  MoveL (T13838) to (110.9, 104.08, 17.5) mm, rotated rx 180 ry 0 rz -180 deg; joints [2.977, 71.493, -37.876, 5.367, -33.733, -4.467]
  MoveL (T13839) to (110.9, 104.08, 15.5) mm, rotated rx 180 ry 0 rz -180 deg; joints [2.977, 71.493, -37.876, 5.367, -33.733, -4.467]
  Set speed (40.0 mm/s)
  Call Extruder 2.0
  MoveL (T13840) to (110.9, 104.08, 15.5) mm, rotated rx 180 ry 0 rz -180 deg; joints [1.43, 67.002, -29.425, 2.343, -37.6, -1.857]
  Set speed (26.9 mm/s)
  MoveL (T13841) to (110.9, 104.08, 15.5) mm, rotated rx 180 ry 0 rz -180 deg; joints [1.43, 67.002, -29.425, 2.343, -37.6, -1.857]
  Call Extruder 0.01643
  MoveL (T13842) to (111.26, 104.43, 15.5) mm, rotated rx 180 ry 0 rz -180 deg; joints [1.43, 67.002, -29.425, 2.343, -37.6, -1.857]
  Call Extruder 0.0201
  MoveL (T13843) to (111.26, 105.05, 15.5) mm, rotated rx 180 ry 0 rz -180 deg; joints [1.431, 66.869, -29.176, 2.34, -37.717, -1.851]
  Call Extruder 0.01643
  MoveL (T13844) to (110.9, 104.69, 15.5) mm, rotated rx 180 ry 0 rz -180 deg; joints [1.431, 66.869, -29.176, 2.34, -37.717, -1.851]
  Set speed (45.0 mm/s)
  Call Extruder -1.6
  MoveL (T13845) to (110.9, 104.69, 15.5) mm, rotated rx 180 ry 0 rz -180 deg; joints [1.431, 66.869, -29.176, 2.34, -37.717, -1.851]
  Set speed (120.0 mm/s)
  MoveL (T13846) to (110.9, 104.69, 15.5) mm, rotated rx 180 ry 0 rz -180 deg; joints [3.031, 71.501, -37.892, 5.464, -33.73, -4.548]
  Call Extruder -0.17945
  MoveL (T13847) to (111.26, 105.05, 15.5) mm, rotated rx 180 ry 0 rz -180 deg; joints [3.031, 71.501, -37.892, 5.464, -33.73, -4.548]
  Call Extruder -0.20055
  MoveL (T13848) to (111.26, 104.49, 15.5) mm, rotated rx 180 ry 0 rz -180 deg; joints [3.031, 71.501, -37.892, 5.464, -33.73, -4.548]
  Set speed (45.0 mm/s)
  Call Extruder -0.02
  MoveL (T13849) to (111.26, 104.49, 15.5) mm, rotated rx 180 ry 0 rz -180 deg; joints [3.084, 71.51, -37.908, 5.56, -33.726, -4.629]
  Set speed (150.0 mm/s)
  MoveL (T13850) to (111.26, 104.49, 17.5) mm, rotated rx 180 ry 0 rz -180 deg; joints [3.084, 71.51, -37.908, 5.56, -33.726, -4.629]
  MoveL (T13851) to (117.12, 105.75, 17.5) mm, rotated rx 180 ry 0 rz -180 deg; joints [1.432, 66.737, -28.928, 2.336, -37.833, -1.845]
  MoveL (T13852) to (117.12, 105.75, 15.5) mm, rotated rx 180 ry 0 rz -180 deg; joints [1.432, 66.737, -28.928, 2.336, -37.833, -1.845]
  Set speed (40.0 mm/s)
  Call Extruder 2.0
  MoveL (T13853) to (117.12, 105.75, 15.5) mm, rotated rx 180 ry 0 rz -180 deg; joints [1.434, 66.606, -28.681, 2.332, -37.949, -1.839]
  Set speed (26.9 mm/s)
  MoveL (T13854) to (117.12, 105.75, 15.5) mm, rotated rx 180 ry 0 rz -180 deg; joints [1.434, 66.606, -28.681, 2.332, -37.949, -1.839]
  Call Extruder 0.01433
  MoveL (T13855) to (117.59, 105.75, 15.5) mm, rotated rx 180 ry 0 rz -180 deg; joints [1.434, 66.606, -28.681, 2.332, -37.949, -1.839]
  Call Extruder 0.05792
  MoveL (T13856) to (117.59, 103.84, 15.5) mm, rotated rx 180 ry 0 rz -180 deg; joints [1.434, 66.606, -28.681, 2.332, -37.949, -1.839]
  Call Extruder 0.00216
  MoveL (T13857) to (117.66, 103.84, 15.5) mm, rotated rx 180 ry 0 rz -180 deg; joints [1.434, 66.606, -28.681, 2.332, -37.949, -1.839]
  Call Extruder 0.10261
  MoveL (T13858) to (120.04, 106.23, 15.5) mm, rotated rx 180 ry 0 rz -180 deg; joints [3.137, 71.518, -37.924, 5.657, -33.723, -4.71]
  Call Extruder 0.0339
  MoveL (T13859) to (121.16, 106.23, 15.5) mm, rotated rx 180 ry 0 rz -180 deg; joints [3.137, 71.518, -37.924, 5.657, -33.723, -4.71]
  Call Extruder 0.07254
  MoveL (T13860) to (121.16, 103.84, 15.5) mm, rotated rx 180 ry 0 rz -180 deg; joints [3.137, 71.518, -37.924, 5.657, -33.723, -4.71]
  Call Extruder 0.7458
  MoveL (T13861) to (103.84, 121.16, 15.5) mm, rotated rx 180 ry 0 rz -180 deg; joints [3.19, 71.527, -37.941, 5.753, -33.72, -4.79]
  Call Extruder 0.10645
  MoveL (T13862) to (103.84, 117.66, 15.5) mm, rotated rx 180 ry 0 rz -180 deg; joints [3.19, 71.527, -37.941, 5.753, -33.72, -4.79]
  Call Extruder 0.15054
  MoveL (T13863) to (107.34, 121.16, 15.5) mm, rotated rx 180 ry 0 rz -180 deg; joints [3.19, 71.527, -37.941, 5.753, -33.72, -4.79]
  Call Extruder 0.03385
  MoveL (T13864) to (108.45, 121.16, 15.5) mm, rotated rx 180 ry 0 rz -180 deg; joints [1.435, 66.475, -28.435, 2.328, -38.064, -1.833]
  Call Extruder 0.45878
  MoveL (T13865) to (119.1, 110.51, 15.5) mm, rotated rx 180 ry 0 rz -180 deg; joints [1.435, 66.475, -28.435, 2.328, -38.064, -1.833]
  Call Extruder 0.00222
  MoveL (T13866) to (119.1, 110.43, 15.5) mm, rotated rx 180 ry 0 rz -180 deg; joints [1.435, 66.475, -28.435, 2.328, -38.064, -1.833]
  Call Extruder 0.00558
  MoveL (T13867) to (119.23, 110.3, 15.5) mm, rotated rx 180 ry 0 rz -180 deg; joints [1.436, 66.41, -28.312, 2.326, -38.121, -1.83]
  Call Extruder 0.00874
  MoveL (T13868) to (119.23, 110.02, 15.5) mm, rotated rx 180 ry 0 rz -180 deg; joints [1.436, 66.41, -28.312, 2.326, -38.121, -1.83]
  Call Extruder 0.18404
  MoveL (T13869) to (114.96, 105.75, 15.5) mm, rotated rx 180 ry 0 rz -180 deg; joints [1.436, 66.41, -28.312, 2.326, -38.121, -1.83]
  Call Extruder 0.00938
  MoveL (T13870) to (114.65, 105.75, 15.5) mm, rotated rx 180 ry 0 rz -180 deg; joints [1.436, 66.41, -28.312, 2.326, -38.121, -1.83]
  Call Extruder 0.46548
  MoveL (T13871) to (103.84, 116.55, 15.5) mm, rotated rx 180 ry 0 rz -180 deg; joints [1.436, 66.41, -28.312, 2.326, -38.121, -1.83]
  Call Extruder 0.10645
  MoveL (T13872) to (103.84, 113.06, 15.5) mm, rotated rx 180 ry 0 rz -180 deg; joints [1.463, 66.412, -28.315, 2.371, -38.12, -1.866]
  Call Extruder 0.34896
  MoveL (T13873) to (111.94, 121.16, 15.5) mm, rotated rx 180 ry 0 rz -180 deg; joints [3.218, 71.452, -37.799, 5.794, -33.788, -4.82]
  Call Extruder 0.03385
  MoveL (T13874) to (113.06, 121.16, 15.5) mm, rotated rx 180 ry 0 rz -180 deg; joints [3.221, 71.293, -37.5, 5.778, -33.928, -4.799]
  Call Extruder 0.26585
  MoveL (T13875) to (119.23, 114.98, 15.5) mm, rotated rx 180 ry 0 rz -180 deg; joints [1.518, 66.415, -28.322, 2.46, -38.119, -1.936]
  Call Extruder 0.01108
  MoveL (T13876) to (119.23, 114.62, 15.5) mm, rotated rx 180 ry 0 rz -180 deg; joints [1.518, 66.415, -28.322, 2.46, -38.119, -1.936]
  Call Extruder 0.38238
  MoveL (T13877) to (110.35, 105.75, 15.5) mm, rotated rx 180 ry 0 rz -180 deg; joints [1.518, 66.415, -28.322, 2.46, -38.119, -1.936]
  Call Extruder 0.00938
  MoveL (T13878) to (110.04, 105.75, 15.5) mm, rotated rx 180 ry 0 rz -180 deg; joints [1.573, 66.419, -28.328, 2.55, -38.118, -2.006]
  Call Extruder 0.26706
  MoveL (T13879) to (103.84, 111.94, 15.5) mm, rotated rx 180 ry 0 rz -180 deg; joints [3.224, 71.135, -37.203, 5.763, -34.067, -4.779]
  Call Extruder 0.07441
  MoveL (T13880) to (103.84, 109.5, 15.5) mm, rotated rx 180 ry 0 rz -180 deg; joints [3.224, 71.135, -37.203, 5.763, -34.067, -4.779]
  Set speed (45.0 mm/s)
  Call Extruder -1.6
  MoveL (T13881) to (103.84, 109.5, 15.5) mm, rotated rx 180 ry 0 rz -180 deg; joints [3.227, 70.978, -36.908, 5.748, -34.205, -4.758]
  Set speed (120.0 mm/s)
  MoveL (T13882) to (103.84, 109.5, 15.5) mm, rotated rx 180 ry 0 rz -180 deg; joints [3.227, 70.978, -36.908, 5.748, -34.205, -4.758]
  Call Extruder -0.38
  MoveL (T13883) to (103.84, 110.57, 15.5) mm, rotated rx 180 ry 0 rz -180 deg; joints [1.629, 66.423, -28.335, 2.639, -38.117, -2.077]
  Set speed (45.0 mm/s)
  Call Extruder -0.02
  MoveL (T13884) to (103.84, 110.57, 15.5) mm, rotated rx 180 ry 0 rz -180 deg; joints [1.629, 66.423, -28.335, 2.639, -38.117, -2.077]
  Set speed (150.0 mm/s)
  MoveL (T13885) to (103.84, 110.57, 17.5) mm, rotated rx 180 ry 0 rz -180 deg; joints [1.684, 66.426, -28.342, 2.728, -38.116, -2.147]
  MoveL (T13886) to (119.1, 110.71, 17.5) mm, rotated rx 180 ry 0 rz -180 deg; joints [1.684, 66.426, -28.342, 2.728, -38.116, -2.147]
  MoveL (T13887) to (119.1, 110.71, 15.5) mm, rotated rx 180 ry 0 rz -180 deg; joints [1.684, 66.426, -28.342, 2.728, -38.116, -2.147]
  Set speed (40.0 mm/s)
  Call Extruder 2.0
  MoveL (T13888) to (119.1, 110.71, 15.5) mm, rotated rx 180 ry 0 rz -180 deg; joints [3.23, 70.823, -36.615, 5.733, -34.342, -4.738]
  Set speed (26.9 mm/s)
  MoveL (T13889) to (119.1, 110.71, 15.5) mm, rotated rx 180 ry 0 rz -180 deg; joints [3.233, 70.668, -36.324, 5.718, -34.477, -4.719]
  Call Extruder 0.00658
  MoveL (T13890) to (119.1, 110.93, 15.5) mm, rotated rx 180 ry 0 rz -180 deg; joints [3.233, 70.668, -36.324, 5.718, -34.477, -4.719]
  Call Extruder 0.01378
  MoveL (T13891) to (119.42, 111.25, 15.5) mm, rotated rx 180 ry 0 rz -180 deg; joints [3.233, 70.668, -36.324, 5.718, -34.477, -4.719]
  Call Extruder 0.03162
  MoveL (T13892) to (120.46, 111.25, 15.5) mm, rotated rx 180 ry 0 rz -180 deg; joints [1.739, 66.43, -28.35, 2.818, -38.114, -2.217]
  Call Extruder 0.03012
  MoveL (T13893) to (121.16, 111.94, 15.5) mm, rotated rx 180 ry 0 rz -180 deg; joints [1.739, 66.43, -28.35, 2.818, -38.114, -2.217]
  Call Extruder 0.02649
  MoveL (T13894) to (121.16, 112.81, 15.5) mm, rotated rx 180 ry 0 rz -180 deg; joints [1.739, 66.43, -28.35, 2.818, -38.114, -2.217]
  Call Extruder 0.04792
  MoveL (T13895) to (119.58, 112.81, 15.5) mm, rotated rx 180 ry 0 rz -180 deg; joints [1.794, 66.434, -28.357, 2.907, -38.113, -2.288]
  Set speed (150.0 mm/s)
  MoveL (T13896) to (120.91, 113.57, 15.5) mm, rotated rx 180 ry 0 rz -180 deg; joints [1.794, 66.434, -28.357, 2.907, -38.113, -2.288]
  Set speed (26.9 mm/s)
  MoveL (T13897) to (120.91, 113.57, 15.5) mm, rotated rx 180 ry 0 rz -180 deg; joints [3.236, 70.515, -36.035, 5.704, -34.612, -4.699]
  Call Extruder 0.01626
  MoveL (T13898) to (120.56, 113.22, 15.5) mm, rotated rx 180 ry 0 rz -180 deg; joints [3.236, 70.515, -36.035, 5.704, -34.612, -4.699]
  Call Extruder 0.02045
  MoveL (T13899) to (119.94, 113.22, 15.5) mm, rotated rx 180 ry 0 rz -180 deg; joints [3.236, 70.515, -36.035, 5.704, -34.612, -4.699]
  Call Extruder 0.01626
  MoveL (T13900) to (120.29, 113.57, 15.5) mm, rotated rx 180 ry 0 rz -180 deg; joints [3.239, 70.362, -35.748, 5.69, -34.746, -4.68]
  Set speed (45.0 mm/s)
  Call Extruder -1.6
  MoveL (T13901) to (120.29, 113.57, 15.5) mm, rotated rx 180 ry 0 rz -180 deg; joints [3.239, 70.362, -35.748, 5.69, -34.746, -4.68]
  Set speed (120.0 mm/s)
  MoveL (T13902) to (120.29, 113.57, 15.5) mm, rotated rx 180 ry 0 rz -180 deg; joints [3.239, 70.362, -35.748, 5.69, -34.746, -4.68]
  Call Extruder -0.17616
  MoveL (T13903) to (119.94, 113.22, 15.5) mm, rotated rx 180 ry 0 rz -180 deg; joints [1.849, 66.438, -28.365, 2.996, -38.111, -2.358]
  Call Extruder -0.20384
  MoveL (T13904) to (120.51, 113.22, 15.5) mm, rotated rx 180 ry 0 rz -180 deg; joints [1.849, 66.438, -28.365, 2.996, -38.111, -2.358]
  Set speed (45.0 mm/s)
  Call Extruder -0.02
  MoveL (T13905) to (120.51, 113.22, 15.5) mm, rotated rx 180 ry 0 rz -180 deg; joints [1.904, 66.443, -28.373, 3.086, -38.11, -2.429]
  Set speed (150.0 mm/s)
  MoveL (T13906) to (120.51, 113.22, 17.5) mm, rotated rx 180 ry 0 rz -180 deg; joints [1.904, 66.443, -28.373, 3.086, -38.11, -2.429]
  MoveL (T13907) to (121.02, 111.02, 17.5) mm, rotated rx 180 ry 0 rz -180 deg; joints [3.242, 70.211, -35.463, 5.676, -34.88, -4.661]
  MoveL (T13908) to (121.02, 111.02, 15.5) mm, rotated rx 180 ry 0 rz -180 deg; joints [3.242, 70.211, -35.463, 5.676, -34.88, -4.661]
  Set speed (40.0 mm/s)
  Call Extruder 2.0
  MoveL (T13909) to (121.02, 111.02, 15.5) mm, rotated rx 180 ry 0 rz -180 deg; joints [3.245, 70.06, -35.18, 5.663, -35.012, -4.643]
  Set speed (26.9 mm/s)
  MoveL (T13910) to (121.02, 111.02, 15.5) mm, rotated rx 180 ry 0 rz -180 deg; joints [3.245, 70.06, -35.18, 5.663, -35.012, -4.643]
  Call Extruder 0.01707
  MoveL (T13911) to (120.64, 110.65, 15.5) mm, rotated rx 180 ry 0 rz -180 deg; joints [1.959, 66.447, -28.381, 3.175, -38.108, -2.499]
  Call Extruder 0.01989
  MoveL (T13912) to (120.03, 110.65, 15.5) mm, rotated rx 180 ry 0 rz -180 deg; joints [1.959, 66.447, -28.381, 3.175, -38.108, -2.499]
  Call Extruder 0.00867
  MoveL (T13913) to (120.22, 110.84, 15.5) mm, rotated rx 180 ry 0 rz -180 deg; joints [2.014, 66.451, -28.39, 3.264, -38.107, -2.57]
  Call Extruder 0.01989
  MoveL (T13914) to (119.61, 110.84, 15.5) mm, rotated rx 180 ry 0 rz -180 deg; joints [2.014, 66.451, -28.39, 3.264, -38.107, -2.57]
  Call Extruder 0.01299
  MoveL (T13915) to (119.32, 110.56, 15.5) mm, rotated rx 180 ry 0 rz -180 deg; joints [2.014, 66.451, -28.39, 3.264, -38.107, -2.57]
  Set speed (45.0 mm/s)
  Call Extruder -1.6
  MoveL (T13916) to (119.32, 110.56, 15.5) mm, rotated rx 180 ry 0 rz -180 deg; joints [3.248, 69.911, -34.899, 5.649, -35.143, -4.625]
  Set speed (120.0 mm/s)
  MoveL (T13917) to (119.32, 110.56, 15.5) mm, rotated rx 180 ry 0 rz -180 deg; joints [3.248, 69.911, -34.899, 5.649, -35.143, -4.625]
  Call Extruder -0.14256
  MoveL (T13918) to (119.61, 110.84, 15.5) mm, rotated rx 180 ry 0 rz -180 deg; joints [3.252, 69.762, -34.619, 5.637, -35.274, -4.607]
  Call Extruder -0.21839
  MoveL (T13919) to (120.22, 110.84, 15.5) mm, rotated rx 180 ry 0 rz -180 deg; joints [2.069, 66.456, -28.398, 3.354, -38.105, -2.64]
  Call Extruder -0.01905
  MoveL (T13920) to (120.18, 110.8, 15.5) mm, rotated rx 180 ry 0 rz -180 deg; joints [2.069, 66.456, -28.398, 3.354, -38.105, -2.64]
  Set speed (45.0 mm/s)
  Call Extruder -0.02
  MoveL (T13921) to (120.18, 110.8, 15.5) mm, rotated rx 180 ry 0 rz -180 deg; joints [2.069, 66.456, -28.398, 3.354, -38.105, -2.64]
  Set speed (150.0 mm/s)
  MoveL (T13922) to (120.18, 110.8, 17.5) mm, rotated rx 180 ry 0 rz -180 deg; joints [2.124, 66.461, -28.407, 3.443, -38.104, -2.711]
  MoveL (T13923) to (104.34, 103.54, 17.5) mm, rotated rx 180 ry 0 rz -180 deg; joints [2.124, 66.461, -28.407, 3.443, -38.104, -2.711]
  MoveL (T13924) to (104.34, 103.54, 15.7) mm, rotated rx 180 ry 0 rz -180 deg; joints [2.124, 66.461, -28.407, 3.443, -38.104, -2.711]
  Set speed (40.0 mm/s)
  Call Extruder 2.0
  MoveL (T13925) to (104.34, 103.54, 15.7) mm, rotated rx 180 ry 0 rz -180 deg; joints [3.255, 69.615, -34.341, 5.624, -35.404, -4.589]
  Set speed (26.8 mm/s)
  MoveL (T13926) to (104.34, 103.54, 15.7) mm, rotated rx 180 ry 0 rz -180 deg; joints [3.258, 69.468, -34.065, 5.611, -35.533, -4.571]
  Call Extruder 0.07908
  MoveL (T13927) to (106.94, 103.54, 15.7) mm, rotated rx 180 ry 0 rz -180 deg; joints [3.258, 69.468, -34.065, 5.611, -35.533, -4.571]
  Call Extruder 0.05792
  MoveL (T13928) to (106.93, 105.44, 15.7) mm, rotated rx 180 ry 0 rz -180 deg; joints [2.179, 66.466, -28.417, 3.533, -38.102, -2.781]
  Call Extruder 0.11363
  MoveL (T13929) to (110.66, 105.44, 15.7) mm, rotated rx 180 ry 0 rz -180 deg; joints [2.179, 66.466, -28.417, 3.533, -38.102, -2.781]
  Call Extruder 0.05792
  MoveL (T13930) to (110.67, 103.54, 15.7) mm, rotated rx 180 ry 0 rz -180 deg; joints [2.234, 66.471, -28.426, 3.622, -38.1, -2.852]
  Call Extruder 0.09209
  MoveL (T13931) to (113.69, 103.54, 15.7) mm, rotated rx 180 ry 0 rz -180 deg; joints [2.234, 66.471, -28.426, 3.622, -38.1, -2.852]
  Call Extruder 0.05792
  MoveL (T13932) to (113.69, 105.44, 15.7) mm, rotated rx 180 ry 0 rz -180 deg; joints [3.261, 69.322, -33.791, 5.599, -35.661, -4.554]
  Call Extruder 0.11347
  MoveL (T13933) to (117.41, 105.44, 15.7) mm, rotated rx 180 ry 0 rz -180 deg; joints [3.261, 69.322, -33.791, 5.599, -35.661, -4.554]
  Call Extruder 0.05792
  MoveL (T13934) to (117.41, 103.54, 15.7) mm, rotated rx 180 ry 0 rz -180 deg; joints [3.261, 69.322, -33.791, 5.599, -35.661, -4.554]
  Call Extruder 0.12333
  MoveL (T13935) to (121.46, 103.54, 15.7) mm, rotated rx 180 ry 0 rz -180 deg; joints [3.264, 69.177, -33.518, 5.587, -35.789, -4.537]
  Call Extruder 0.08749
  MoveL (T13936) to (121.46, 106.41, 15.7) mm, rotated rx 180 ry 0 rz -180 deg; joints [3.264, 69.177, -33.518, 5.587, -35.789, -4.537]
  Call Extruder 0.05864
  MoveL (T13937) to (119.54, 106.41, 15.7) mm, rotated rx 180 ry 0 rz -180 deg; joints [2.289, 66.476, -28.436, 3.712, -38.099, -2.922]
  Call Extruder 0.11623
  MoveL (T13938) to (119.53, 110.23, 15.7) mm, rotated rx 180 ry 0 rz -180 deg; joints [2.289, 66.476, -28.436, 3.712, -38.099, -2.922]
  Call Extruder 0.05869
  MoveL (T13939) to (121.46, 110.23, 15.7) mm, rotated rx 180 ry 0 rz -180 deg; joints [2.344, 66.481, -28.446, 3.801, -38.097, -2.993]
  Call Extruder 0.10898
  MoveL (T13940) to (121.46, 113.8, 15.7) mm, rotated rx 180 ry 0 rz -180 deg; joints [3.267, 69.033, -33.247, 5.575, -35.915, -4.52]
  Call Extruder 0.05874
  MoveL (T13941) to (119.53, 113.8, 15.7) mm, rotated rx 180 ry 0 rz -180 deg; joints [3.267, 69.033, -33.247, 5.575, -35.915, -4.52]
  Call Extruder 0.11558
  MoveL (T13942) to (119.53, 117.59, 15.7) mm, rotated rx 180 ry 0 rz -180 deg; joints [3.27, 68.89, -32.977, 5.563, -36.041, -4.503]
  Call Extruder 0.05879
  MoveL (T13943) to (121.46, 117.6, 15.7) mm, rotated rx 180 ry 0 rz -180 deg; joints [3.27, 68.89, -32.977, 5.563, -36.041, -4.503]
  Call Extruder 0.11768
  MoveL (T13944) to (121.46, 121.46, 15.7) mm, rotated rx 180 ry 0 rz -180 deg; joints [3.27, 68.89, -32.977, 5.563, -36.041, -4.503]
  Call Extruder 0.54596
  MoveL (T13945) to (103.54, 121.46, 15.7) mm, rotated rx 180 ry 0 rz -180 deg; joints [2.399, 66.487, -28.456, 3.89, -38.095, -3.064]
  Call Extruder 0.54596
  MoveL (T13946) to (103.54, 103.54, 15.7) mm, rotated rx 180 ry 0 rz -180 deg; joints [2.399, 66.487, -28.456, 3.89, -38.095, -3.064]
  Call Extruder 0.02254
  MoveL (T13947) to (104.28, 103.54, 15.7) mm, rotated rx 180 ry 0 rz -180 deg; joints [2.454, 66.492, -28.466, 3.98, -38.093, -3.134]
  Set speed (150.0 mm/s)
  MoveL (T13948) to (103.53, 103.13, 15.7) mm, rotated rx 180 ry 0 rz -180 deg; joints [2.454, 66.492, -28.466, 3.98, -38.093, -3.134]
  Set speed (26.8 mm/s)
  MoveL (T13949) to (103.53, 103.13, 15.7) mm, rotated rx 180 ry 0 rz -180 deg; joints [2.454, 66.492, -28.466, 3.98, -38.093, -3.134]
  Call Extruder 0.11607
  MoveL (T13950) to (107.34, 103.13, 15.7) mm, rotated rx 180 ry 0 rz -180 deg; joints [3.273, 68.747, -32.709, 5.552, -36.166, -4.487]
  Call Extruder 0.05792
  MoveL (T13951) to (107.34, 105.03, 15.7) mm, rotated rx 180 ry 0 rz -180 deg; joints [3.273, 68.747, -32.709, 5.552, -36.166, -4.487]
  Call Extruder 0.08883
  MoveL (T13952) to (110.26, 105.03, 15.7) mm, rotated rx 180 ry 0 rz -180 deg; joints [3.273, 68.747, -32.709, 5.552, -36.166, -4.487]
  Call Extruder 0.05792
  MoveL (T13953) to (110.26, 103.13, 15.7) mm, rotated rx 180 ry 0 rz -180 deg; joints [3.276, 68.606, -32.443, 5.541, -36.291, -4.471]
  Call Extruder 0.11688
  MoveL (T13954) to (114.09, 103.13, 15.7) mm, rotated rx 180 ry 0 rz -180 deg; joints [3.276, 68.606, -32.443, 5.541, -36.291, -4.471]
  Call Extruder 0.05792
  MoveL (T13955) to (114.1, 105.03, 15.7) mm, rotated rx 180 ry 0 rz -180 deg; joints [3.276, 68.606, -32.443, 5.541, -36.291, -4.471]
  Call Extruder 0.08867
  MoveL (T13956) to (117.01, 105.03, 15.7) mm, rotated rx 180 ry 0 rz -180 deg; joints [2.509, 66.498, -28.477, 4.069, -38.091, -3.205]
  Call Extruder 0.05792
  MoveL (T13957) to (117, 103.13, 15.7) mm, rotated rx 180 ry 0 rz -180 deg; joints [2.509, 66.498, -28.477, 4.069, -38.091, -3.205]
  Call Extruder 0.14814
  MoveL (T13958) to (121.87, 103.13, 15.7) mm, rotated rx 180 ry 0 rz -180 deg; joints [2.509, 66.498, -28.477, 4.069, -38.091, -3.205]
  Call Extruder 0.11229
  MoveL (T13959) to (121.87, 106.82, 15.7) mm, rotated rx 180 ry 0 rz -180 deg; joints [2.564, 66.504, -28.488, 4.159, -38.089, -3.275]
  Call Extruder 0.05865
  MoveL (T13960) to (119.94, 106.82, 15.7) mm, rotated rx 180 ry 0 rz -180 deg; joints [2.564, 66.504, -28.488, 4.159, -38.089, -3.275]
  Call Extruder 0.09143
  MoveL (T13961) to (119.94, 109.82, 15.7) mm, rotated rx 180 ry 0 rz -180 deg; joints [3.279, 68.465, -32.178, 5.53, -36.415, -4.455]
  Call Extruder 0.05869
  MoveL (T13962) to (121.87, 109.82, 15.7) mm, rotated rx 180 ry 0 rz -180 deg; joints [3.279, 68.465, -32.178, 5.53, -36.415, -4.455]
  Call Extruder 0.13381
  MoveL (T13963) to (121.87, 114.21, 15.7) mm, rotated rx 180 ry 0 rz -180 deg; joints [3.279, 68.465, -32.178, 5.53, -36.415, -4.455]
  Call Extruder 0.05875
  MoveL (T13964) to (119.94, 114.21, 15.7) mm, rotated rx 180 ry 0 rz -180 deg; joints [3.282, 68.325, -31.914, 5.519, -36.538, -4.439]
  Call Extruder 0.09077
  MoveL (T13965) to (119.94, 117.19, 15.7) mm, rotated rx 180 ry 0 rz -180 deg; joints [3.282, 68.325, -31.914, 5.519, -36.538, -4.439]
  Call Extruder 0.05879
  MoveL (T13966) to (121.87, 117.19, 15.7) mm, rotated rx 180 ry 0 rz -180 deg; joints [3.282, 68.325, -31.914, 5.519, -36.538, -4.439]
  Call Extruder 0.14247
  MoveL (T13967) to (121.87, 121.87, 15.7) mm, rotated rx 180 ry 0 rz -180 deg; joints [2.619, 66.509, -28.499, 4.248, -38.087, -3.346]
  Call Extruder 0.57077
  MoveL (T13968) to (103.13, 121.87, 15.7) mm, rotated rx 180 ry 0 rz -180 deg; joints [2.619, 66.509, -28.499, 4.248, -38.087, -3.346]
  Call Extruder 0.57077
  MoveL (T13969) to (103.13, 103.13, 15.7) mm, rotated rx 180 ry 0 rz -180 deg; joints [2.674, 66.516, -28.51, 4.338, -38.085, -3.417]
  Call Extruder 0.01036
  MoveL (T13970) to (103.47, 103.13, 15.7) mm, rotated rx 180 ry 0 rz -180 deg; joints [2.674, 66.516, -28.51, 4.338, -38.085, -3.417]
  Set speed (150.0 mm/s)
  MoveL (T13971) to (102.72, 102.81, 15.7) mm, rotated rx 180 ry 0 rz -180 deg; joints [3.285, 68.186, -31.652, 5.508, -36.66, -4.423]
  Set speed (25.0 mm/s)
  MoveL (T13972) to (102.72, 102.81, 15.7) mm, rotated rx 180 ry 0 rz -180 deg; joints [3.285, 68.186, -31.652, 5.508, -36.66, -4.423]
  Call Extruder 0.00259
  MoveL (T13973) to (102.72, 102.72, 15.7) mm, rotated rx 180 ry 0 rz -180 deg; joints [3.289, 68.047, -31.392, 5.498, -36.782, -4.408]
  Call Extruder 0.15306
  MoveL (T13974) to (107.75, 102.72, 15.7) mm, rotated rx 180 ry 0 rz -180 deg; joints [3.289, 68.047, -31.392, 5.498, -36.782, -4.408]
  Call Extruder 0.05792
  MoveL (T13975) to (107.75, 104.63, 15.7) mm, rotated rx 180 ry 0 rz -180 deg; joints [2.729, 66.522, -28.522, 4.427, -38.083, -3.488]
  Call Extruder 0.06403
  MoveL (T13976) to (109.85, 104.63, 15.7) mm, rotated rx 180 ry 0 rz -180 deg; joints [2.784, 66.528, -28.534, 4.517, -38.081, -3.558]
  Call Extruder 0.05792
  MoveL (T13977) to (109.85, 102.72, 15.7) mm, rotated rx 180 ry 0 rz -180 deg; joints [2.784, 66.528, -28.534, 4.517, -38.081, -3.558]
  Call Extruder 0.14167
  MoveL (T13978) to (114.5, 102.72, 15.7) mm, rotated rx 180 ry 0 rz -180 deg; joints [2.784, 66.528, -28.534, 4.517, -38.081, -3.558]
  Call Extruder 0.05792
  MoveL (T13979) to (114.5, 104.63, 15.7) mm, rotated rx 180 ry 0 rz -180 deg; joints [3.292, 67.909, -31.132, 5.487, -36.903, -4.393]
  Call Extruder 0.06386
  MoveL (T13980) to (116.6, 104.63, 15.7) mm, rotated rx 180 ry 0 rz -180 deg; joints [3.292, 67.909, -31.132, 5.487, -36.903, -4.393]
  Call Extruder 0.05792
  MoveL (T13981) to (116.6, 102.72, 15.7) mm, rotated rx 180 ry 0 rz -180 deg; joints [3.295, 67.772, -30.875, 5.477, -37.024, -4.378]
  Call Extruder 0.17294
  MoveL (T13982) to (122.28, 102.72, 15.7) mm, rotated rx 180 ry 0 rz -180 deg; joints [3.295, 67.772, -30.875, 5.477, -37.024, -4.378]
  Call Extruder 0.13709
  MoveL (T13983) to (122.28, 107.22, 15.7) mm, rotated rx 180 ry 0 rz -180 deg; joints [3.295, 67.772, -30.875, 5.477, -37.024, -4.378]
  Call Extruder 0.05865
  MoveL (T13984) to (120.35, 107.23, 15.7) mm, rotated rx 180 ry 0 rz -180 deg; joints [2.839, 66.534, -28.546, 4.606, -38.079, -3.629]
  Call Extruder 0.06663
  MoveL (T13985) to (120.35, 109.41, 15.7) mm, rotated rx 180 ry 0 rz -180 deg; joints [2.839, 66.534, -28.546, 4.606, -38.079, -3.629]
  Call Extruder 0.05868
  MoveL (T13986) to (122.28, 109.41, 15.7) mm, rotated rx 180 ry 0 rz -180 deg; joints [2.894, 66.541, -28.558, 4.696, -38.076, -3.7]
  Call Extruder 0.15863
  MoveL (T13987) to (122.28, 114.62, 15.7) mm, rotated rx 180 ry 0 rz -180 deg; joints [2.894, 66.541, -28.558, 4.696, -38.076, -3.7]
  Call Extruder 0.05875
  MoveL (T13988) to (120.35, 114.62, 15.7) mm, rotated rx 180 ry 0 rz -180 deg; joints [3.298, 67.636, -30.618, 5.467, -37.144, -4.363]
  Call Extruder 0.06597
  MoveL (T13989) to (120.34, 116.78, 15.7) mm, rotated rx 180 ry 0 rz -180 deg; joints [3.298, 67.636, -30.618, 5.467, -37.144, -4.363]
  Call Extruder 0.05878
  MoveL (T13990) to (122.28, 116.78, 15.7) mm, rotated rx 180 ry 0 rz -180 deg; joints [3.301, 67.5, -30.363, 5.457, -37.263, -4.348]
  Call Extruder 0.16725
  MoveL (T13991) to (122.28, 122.28, 15.7) mm, rotated rx 180 ry 0 rz -180 deg; joints [3.301, 67.5, -30.363, 5.457, -37.263, -4.348]
  Call Extruder 0.59557
  MoveL (T13992) to (102.72, 122.28, 15.7) mm, rotated rx 180 ry 0 rz -180 deg; joints [3.301, 67.5, -30.363, 5.457, -37.263, -4.348]
  Call Extruder 0.59115
  MoveL (T13993) to (102.72, 102.87, 15.7) mm, rotated rx 180 ry 0 rz -180 deg; joints [2.949, 66.548, -28.57, 4.786, -38.074, -3.771]
  Set speed (150.0 mm/s)
  MoveL (T13994) to (102.78, 102.75, 15.7) mm, rotated rx 180 ry 0 rz -180 deg; joints [2.949, 66.548, -28.57, 4.786, -38.074, -3.771]
  Set speed (45.0 mm/s)
  Call Extruder -1.6
  MoveL (T13995) to (102.78, 102.75, 15.7) mm, rotated rx 180 ry 0 rz -180 deg; joints [2.949, 66.548, -28.57, 4.786, -38.074, -3.771]
  Set speed (120.0 mm/s)
  MoveL (T13996) to (102.78, 102.75, 15.7) mm, rotated rx 180 ry 0 rz -180 deg; joints [3.004, 66.554, -28.583, 4.875, -38.072, -3.841]
  Call Extruder -0.05166
  MoveL (T13997) to (102.72, 102.72, 15.7) mm, rotated rx 180 ry 0 rz -180 deg; joints [3.004, 66.554, -28.583, 4.875, -38.072, -3.841]
  Call Extruder -0.32834
  MoveL (T13998) to (103.65, 102.72, 15.7) mm, rotated rx 180 ry 0 rz -180 deg; joints [3.004, 66.554, -28.583, 4.875, -38.072, -3.841]
  Set speed (45.0 mm/s)
  Call Extruder -0.02
  MoveL (T13999) to (103.65, 102.72, 15.7) mm, rotated rx 180 ry 0 rz -180 deg; joints [3.304, 67.365, -30.109, 5.448, -37.381, -4.334]
  Set speed (150.0 mm/s)
  MoveL (T14000) to (103.65, 102.72, 17.7) mm, rotated rx 180 ry 0 rz -180 deg; joints [3.307, 67.231, -29.857, 5.438, -37.499, -4.319]
  MoveL (T14001) to (106.29, 103.84, 17.7) mm, rotated rx 180 ry 0 rz -180 deg; joints [3.307, 67.231, -29.857, 5.438, -37.499, -4.319]
  MoveL (T14002) to (106.29, 103.84, 15.7) mm, rotated rx 180 ry 0 rz -180 deg; joints [3.059, 66.561, -28.596, 4.965, -38.07, -3.912]
  Set speed (40.0 mm/s)
  Call Extruder 2.0
  MoveL (T14003) to (106.29, 103.84, 15.7) mm, rotated rx 180 ry 0 rz -180 deg; joints [3.059, 66.561, -28.596, 4.965, -38.07, -3.912]
  Set speed (26.8 mm/s)
  MoveL (T14004) to (106.29, 103.84, 15.7) mm, rotated rx 180 ry 0 rz -180 deg; joints [3.059, 66.561, -28.596, 4.965, -38.07, -3.912]
  Call Extruder 0.07441
  MoveL (T14005) to (103.84, 103.84, 15.7) mm, rotated rx 180 ry 0 rz -180 deg; joints [3.114, 66.568, -28.61, 5.054, -38.067, -3.983]
  Call Extruder 0.7458
  MoveL (T14006) to (121.16, 121.16, 15.7) mm, rotated rx 180 ry 0 rz -180 deg; joints [3.114, 66.568, -28.61, 5.054, -38.067, -3.983]
  Call Extruder 0.09909
  MoveL (T14007) to (121.16, 117.9, 15.7) mm, rotated rx 180 ry 0 rz -180 deg; joints [3.311, 67.098, -29.605, 5.429, -37.617, -4.305]
  Call Extruder 0.00735
  MoveL (T14008) to (120.91, 117.9, 15.7) mm, rotated rx 180 ry 0 rz -180 deg; joints [3.311, 67.098, -29.605, 5.429, -37.617, -4.305]
  Call Extruder 0.14015
  MoveL (T14009) to (117.66, 121.16, 15.7) mm, rotated rx 180 ry 0 rz -180 deg; joints [3.311, 67.098, -29.605, 5.429, -37.617, -4.305]
  Call Extruder 0.03385
  MoveL (T14010) to (116.55, 121.16, 15.7) mm, rotated rx 180 ry 0 rz -180 deg; joints [3.314, 66.965, -29.355, 5.42, -37.734, -4.291]
  Call Extruder 0.54738
  MoveL (T14011) to (103.84, 108.45, 15.7) mm, rotated rx 180 ry 0 rz -180 deg; joints [3.314, 66.965, -29.355, 5.42, -37.734, -4.291]
  Call Extruder 0.03385
  MoveL (T14012) to (103.84, 107.34, 15.7) mm, rotated rx 180 ry 0 rz -180 deg; joints [3.314, 66.965, -29.355, 5.42, -37.734, -4.291]
  Call Extruder 0.11997
  MoveL (T14013) to (106.63, 104.55, 15.7) mm, rotated rx 180 ry 0 rz -180 deg; joints [3.169, 66.576, -28.623, 5.144, -38.065, -4.054]
  Call Extruder 0.0363
  MoveL (T14014) to (106.63, 105.75, 15.7) mm, rotated rx 180 ry 0 rz -180 deg; joints [3.169, 66.576, -28.623, 5.144, -38.065, -4.054]
  Call Extruder 0.03811
  MoveL (T14015) to (107.88, 105.75, 15.7) mm, rotated rx 180 ry 0 rz -180 deg; joints [3.169, 66.576, -28.623, 5.144, -38.065, -4.054]
  Set speed (45.0 mm/s)
  Call Extruder -1.6
  MoveL (T14016) to (107.88, 105.75, 15.7) mm, rotated rx 180 ry 0 rz -180 deg; joints [3.224, 66.583, -28.637, 5.234, -38.062, -4.125]
  Set speed (120.0 mm/s)
  MoveL (T14017) to (107.88, 105.75, 15.7) mm, rotated rx 180 ry 0 rz -180 deg; joints [3.224, 66.583, -28.637, 5.234, -38.062, -4.125]
  Call Extruder -0.38
  MoveL (T14018) to (106.81, 105.75, 15.7) mm, rotated rx 180 ry 0 rz -180 deg; joints [3.224, 66.583, -28.637, 5.234, -38.062, -4.125]
  Set speed (45.0 mm/s)
  Call Extruder -0.02
  MoveL (T14019) to (106.81, 105.75, 15.7) mm, rotated rx 180 ry 0 rz -180 deg; joints [3.317, 66.833, -29.107, 5.411, -37.85, -4.277]
  Set speed (150.0 mm/s)
  MoveL (T14020) to (106.81, 105.75, 17.7) mm, rotated rx 180 ry 0 rz -180 deg; joints [3.317, 66.833, -29.107, 5.411, -37.85, -4.277]
  MoveL (T14021) to (110.61, 105.75, 17.7) mm, rotated rx 180 ry 0 rz -180 deg; joints [3.317, 66.833, -29.107, 5.411, -37.85, -4.277]
  MoveL (T14022) to (110.61, 105.75, 15.7) mm, rotated rx 180 ry 0 rz -180 deg; joints [3.317, 66.833, -29.107, 5.411, -37.85, -4.277]
  Set speed (40.0 mm/s)
  Call Extruder 2.0
  MoveL (T14023) to (110.61, 105.75, 15.7) mm, rotated rx 180 ry 0 rz -180 deg; joints [3.32, 66.701, -28.859, 5.402, -37.966, -4.264]
  Set speed (26.8 mm/s)
  MoveL (T14024) to (110.61, 105.75, 15.7) mm, rotated rx 180 ry 0 rz -180 deg; joints [3.32, 66.701, -28.859, 5.402, -37.966, -4.264]
  Call Extruder 0.00593
  MoveL (T14025) to (110.75, 105.87, 15.7) mm, rotated rx 180 ry 0 rz -180 deg; joints [3.262, 66.547, -28.569, 5.292, -38.097, -4.169]
  Call Extruder 0.01451
  MoveL (T14026) to (111.23, 105.87, 15.7) mm, rotated rx 180 ry 0 rz -180 deg; joints [3.262, 66.547, -28.569, 5.292, -38.097, -4.169]
  Call Extruder 0.01375
  MoveL (T14027) to (111.55, 105.55, 15.7) mm, rotated rx 180 ry 0 rz -180 deg; joints [3.262, 66.547, -28.569, 5.292, -38.097, -4.169]
  Call Extruder 0.04007
  MoveL (T14028) to (111.55, 104.24, 15.7) mm, rotated rx 180 ry 0 rz -180 deg; joints [3.262, 66.547, -28.569, 5.292, -38.097, -4.169]
  Call Extruder 0.01698
  MoveL (T14029) to (111.94, 103.84, 15.7) mm, rotated rx 180 ry 0 rz -180 deg; joints [3.262, 66.547, -28.569, 5.292, -38.097, -4.169]
  Call Extruder 0.02453
  MoveL (T14030) to (112.75, 103.84, 15.7) mm, rotated rx 180 ry 0 rz -180 deg; joints [3.262, 66.547, -28.569, 5.292, -38.097, -4.169]
  Call Extruder 0.04988
  MoveL (T14031) to (112.75, 105.48, 15.7) mm, rotated rx 180 ry 0 rz -180 deg; joints [3.262, 66.547, -28.569, 5.292, -38.097, -4.169]
  Set speed (150.0 mm/s)
  MoveL (T14032) to (113.57, 104.67, 15.7) mm, rotated rx 180 ry 0 rz -180 deg; joints [3.262, 66.547, -28.569, 5.292, -38.097, -4.169]
  Set speed (26.8 mm/s)
  MoveL (T14033) to (113.57, 104.67, 15.7) mm, rotated rx 180 ry 0 rz -180 deg; joints [3.262, 66.547, -28.569, 5.292, -38.097, -4.169]
  Call Extruder 0.01928
  MoveL (T14034) to (113.16, 105.08, 15.7) mm, rotated rx 180 ry 0 rz -180 deg; joints [3.32, 66.701, -28.859, 5.402, -37.966, -4.264]
  Call Extruder 0.02098
  MoveL (T14035) to (113.16, 104.45, 15.7) mm, rotated rx 180 ry 0 rz -180 deg; joints [3.32, 66.701, -28.859, 5.402, -37.966, -4.264]
  Call Extruder 0.01928
  MoveL (T14036) to (113.57, 104.05, 15.7) mm, rotated rx 180 ry 0 rz -180 deg; joints [3.318, 66.77, -28.989, 5.407, -37.905, -4.271]
  Set speed (45.0 mm/s)
  Call Extruder -1.6
  MoveL (T14037) to (113.57, 104.05, 15.7) mm, rotated rx 180 ry 0 rz -180 deg; joints [3.318, 66.77, -28.989, 5.407, -37.905, -4.271]
  Set speed (120.0 mm/s)
  MoveL (T14038) to (113.57, 104.05, 15.7) mm, rotated rx 180 ry 0 rz -180 deg; joints [3.318, 66.77, -28.989, 5.407, -37.905, -4.271]
  Call Extruder -0.20613
  MoveL (T14039) to (113.16, 104.45, 15.7) mm, rotated rx 180 ry 0 rz -180 deg; joints [3.318, 66.77, -28.989, 5.407, -37.905, -4.271]
  Call Extruder -0.17387
  MoveL (T14040) to (113.16, 104.94, 15.7) mm, rotated rx 180 ry 0 rz -180 deg; joints [3.318, 66.77, -28.989, 5.407, -37.905, -4.271]
  Set speed (45.0 mm/s)
  Call Extruder -0.02
  MoveL (T14041) to (113.16, 104.94, 15.7) mm, rotated rx 180 ry 0 rz -180 deg; joints [3.318, 66.77, -28.989, 5.407, -37.905, -4.271]
  Set speed (150.0 mm/s)
  MoveL (T14042) to (113.16, 104.94, 17.7) mm, rotated rx 180 ry 0 rz -180 deg; joints [3.318, 66.77, -28.989, 5.407, -37.905, -4.271]
  MoveL (T14043) to (110.86, 105.65, 17.7) mm, rotated rx 180 ry 0 rz -180 deg; joints [3.318, 66.532, -28.948, 5.431, -37.709, -4.301]
  MoveL (T14044) to (110.86, 105.65, 15.7) mm, rotated rx 180 ry 0 rz -180 deg; joints [3.318, 66.532, -28.948, 5.431, -37.709, -4.301]
  Set speed (40.0 mm/s)
  Call Extruder 2.0
  MoveL (T14045) to (110.86, 105.65, 15.7) mm, rotated rx 180 ry 0 rz -180 deg; joints [3.318, 66.532, -28.948, 5.431, -37.709, -4.301]
  Set speed (26.8 mm/s)
  MoveL (T14046) to (110.86, 105.65, 15.7) mm, rotated rx 180 ry 0 rz -180 deg; joints [3.318, 66.532, -28.948, 5.431, -37.709, -4.301]
  Call Extruder 0.01251
  MoveL (T14047) to (111.14, 105.37, 15.7) mm, rotated rx 180 ry 0 rz -180 deg; joints [3.318, 66.532, -28.948, 5.431, -37.709, -4.301]
  Call Extruder 0.01919
  MoveL (T14048) to (111.14, 104.77, 15.7) mm, rotated rx 180 ry 0 rz -180 deg; joints [3.318, 66.532, -28.948, 5.431, -37.709, -4.301]
  Call Extruder 0.00781
  MoveL (T14049) to (110.97, 104.94, 15.7) mm, rotated rx 180 ry 0 rz -180 deg; joints [3.82, 66.607, -29.089, 6.256, -37.683, -4.959]
  Call Extruder 0.01919
  MoveL (T14050) to (110.97, 104.34, 15.7) mm, rotated rx 180 ry 0 rz -180 deg; joints [3.82, 66.821, -29.126, 6.231, -37.86, -4.927]
  Call Extruder 0.01606
  MoveL (T14051) to (111.33, 103.98, 15.7) mm, rotated rx 180 ry 0 rz -180 deg; joints [3.82, 66.821, -29.126, 6.231, -37.86, -4.927]
  Set speed (45.0 mm/s)
  Call Extruder -1.6
  MoveL (T14052) to (111.33, 103.98, 15.7) mm, rotated rx 180 ry 0 rz -180 deg; joints [3.82, 66.821, -29.126, 6.231, -37.86, -4.927]
  Set speed (120.0 mm/s)
  MoveL (T14053) to (111.33, 103.98, 15.7) mm, rotated rx 180 ry 0 rz -180 deg; joints [3.82, 66.821, -29.126, 6.231, -37.86, -4.927]
  Call Extruder -0.17962
  MoveL (T14054) to (110.97, 104.34, 15.7) mm, rotated rx 180 ry 0 rz -180 deg; joints [3.82, 66.821, -29.126, 6.231, -37.86, -4.927]
  Call Extruder -0.20038
  MoveL (T14055) to (110.97, 104.9, 15.7) mm, rotated rx 180 ry 0 rz -180 deg; joints [3.82, 66.821, -29.126, 6.231, -37.86, -4.927]
  Set speed (45.0 mm/s)
  Call Extruder -0.02
  MoveL (T14056) to (110.97, 104.9, 15.7) mm, rotated rx 180 ry 0 rz -180 deg; joints [3.82, 66.821, -29.126, 6.231, -37.86, -4.927]
  Set speed (150.0 mm/s)
  MoveL (T14057) to (110.97, 104.9, 17.7) mm, rotated rx 180 ry 0 rz -180 deg; joints [3.82, 66.821, -29.126, 6.231, -37.86, -4.927]
  MoveL (T14058) to (117.12, 105.75, 17.7) mm, rotated rx 180 ry 0 rz -180 deg; joints [3.82, 66.821, -29.126, 6.231, -37.86, -4.927]
  MoveL (T14059) to (117.12, 105.75, 15.7) mm, rotated rx 180 ry 0 rz -180 deg; joints [3.82, 66.821, -29.126, 6.231, -37.86, -4.927]
  Set speed (40.0 mm/s)
  Call Extruder 2.0
  MoveL (T14060) to (117.12, 105.75, 15.7) mm, rotated rx 180 ry 0 rz -180 deg; joints [3.834, 66.317, -28.177, 6.193, -38.303, -4.867]
  Set speed (26.8 mm/s)
  MoveL (T14061) to (117.12, 105.75, 15.7) mm, rotated rx 180 ry 0 rz -180 deg; joints [3.834, 66.317, -28.177, 6.193, -38.303, -4.867]
  Call Extruder 0.01822
  MoveL (T14062) to (117.72, 105.75, 15.7) mm, rotated rx 180 ry 0 rz -180 deg; joints [3.803, 65.911, -27.413, 6.095, -38.656, -4.766]
  Call Extruder 0.05619
  MoveL (T14063) to (117.72, 103.9, 15.7) mm, rotated rx 180 ry 0 rz -180 deg; joints [3.803, 65.911, -27.413, 6.095, -38.656, -4.766]
  Call Extruder 0.09501
  MoveL (T14064) to (119.92, 106.11, 15.7) mm, rotated rx 180 ry 0 rz -180 deg; joints [3.803, 65.911, -27.413, 6.095, -38.656, -4.766]
  Call Extruder 0.03754
  MoveL (T14065) to (121.16, 106.11, 15.7) mm, rotated rx 180 ry 0 rz -180 deg; joints [3.693, 65.591, -26.813, 5.883, -38.926, -4.583]
  Call Extruder 0.0689
  MoveL (T14066) to (121.16, 103.84, 15.7) mm, rotated rx 180 ry 0 rz -180 deg; joints [3.693, 65.591, -26.813, 5.883, -38.926, -4.583]
  Call Extruder 0.7458
  MoveL (T14067) to (103.84, 121.16, 15.7) mm, rotated rx 180 ry 0 rz -180 deg; joints [3.693, 65.591, -26.813, 5.883, -38.926, -4.583]
  Call Extruder 0.10645
  MoveL (T14068) to (103.84, 117.66, 15.7) mm, rotated rx 180 ry 0 rz -180 deg; joints [3.493, 65.421, -26.492, 5.548, -39.06, -4.313]
  Call Extruder 0.15054
  MoveL (T14069) to (107.34, 121.16, 15.7) mm, rotated rx 180 ry 0 rz -180 deg; joints [3.493, 65.421, -26.492, 5.548, -39.06, -4.313]
  Call Extruder 0.03385
  MoveL (T14070) to (108.45, 121.16, 15.7) mm, rotated rx 180 ry 0 rz -180 deg; joints [1.308, 65.214, -26.103, 2.072, -39.129, -1.608]
  Call Extruder 0.45879
  MoveL (T14071) to (119.1, 110.51, 15.7) mm, rotated rx 180 ry 0 rz -180 deg; joints [1.308, 65.214, -26.103, 2.072, -39.129, -1.608]
  Call Extruder 0.00577
  MoveL (T14072) to (119.1, 110.32, 15.7) mm, rotated rx 180 ry 0 rz -180 deg; joints [1.134, 65.303, -26.27, 1.801, -39.046, -1.399]
  Call Extruder 0.00558
  MoveL (T14073) to (119.23, 110.19, 15.7) mm, rotated rx 180 ry 0 rz -180 deg; joints [1, 65.567, -26.767, 1.596, -38.811, -1.244]
  Call Extruder 0.00516
  MoveL (T14074) to (119.23, 110.02, 15.7) mm, rotated rx 180 ry 0 rz -180 deg; joints [1, 65.567, -26.767, 1.596, -38.811, -1.244]
  Call Extruder 0.18405
  MoveL (T14075) to (114.96, 105.75, 15.7) mm, rotated rx 180 ry 0 rz -180 deg; joints [1, 65.567, -26.767, 1.596, -38.811, -1.244]
  Call Extruder 0.00939
  MoveL (T14076) to (114.65, 105.75, 15.7) mm, rotated rx 180 ry 0 rz -180 deg; joints [0.934, 66.034, -27.646, 1.505, -38.398, -1.179]
  Call Extruder 0.46547
  MoveL (T14077) to (103.84, 116.55, 15.7) mm, rotated rx 180 ry 0 rz -180 deg; joints [0.934, 66.034, -27.646, 1.505, -38.398, -1.179]
  Call Extruder 0.10645
  MoveL (T14078) to (103.84, 113.06, 15.7) mm, rotated rx 180 ry 0 rz -180 deg; joints [0.934, 66.034, -27.646, 1.505, -38.398, -1.179]
  Call Extruder 0.34896
  MoveL (T14079) to (111.94, 121.16, 15.7) mm, rotated rx 180 ry 0 rz -180 deg; joints [0.9, 71.665, -38.239, 1.634, -33.436, -1.364]
  Call Extruder 0.03385
  MoveL (T14080) to (113.06, 121.16, 15.7) mm, rotated rx 180 ry 0 rz -180 deg; joints [0.9, 71.665, -38.239, 1.634, -33.436, -1.364]
  Call Extruder 0.26587
  MoveL (T14081) to (119.23, 114.98, 15.7) mm, rotated rx 180 ry 0 rz -180 deg; joints [0.939, 72.175, -39.199, 1.725, -32.988, -1.447]
  Call Extruder 0.01106
  MoveL (T14082) to (119.23, 114.62, 15.7) mm, rotated rx 180 ry 0 rz -180 deg; joints [0.939, 72.175, -39.199, 1.725, -32.988, -1.447]
  Call Extruder 0.38238
  MoveL (T14083) to (110.35, 105.75, 15.7) mm, rotated rx 180 ry 0 rz -180 deg; joints [1.05, 72.578, -39.958, 1.948, -32.635, -1.641]
  Call Extruder 0.00939
  MoveL (T14084) to (110.04, 105.75, 15.7) mm, rotated rx 180 ry 0 rz -180 deg; joints [1.05, 72.578, -39.958, 1.948, -32.635, -1.641]
  Call Extruder 0.26705
  MoveL (T14085) to (103.84, 111.94, 15.7) mm, rotated rx 180 ry 0 rz -180 deg; joints [1.244, 72.781, -40.34, 2.318, -32.462, -1.956]
  Call Extruder 0.07441
  MoveL (T14086) to (103.84, 109.5, 15.7) mm, rotated rx 180 ry 0 rz -180 deg; joints [1.244, 72.781, -40.34, 2.318, -32.462, -1.956]
  Set speed (45.0 mm/s)
  Call Extruder -1.6
  MoveL (T14087) to (103.84, 109.5, 15.7) mm, rotated rx 180 ry 0 rz -180 deg; joints [3.323, 73.051, -40.847, 6.219, -32.356, -5.259]
  Set speed (120.0 mm/s)
  MoveL (T14088) to (103.84, 109.5, 15.7) mm, rotated rx 180 ry 0 rz -180 deg; joints [3.323, 73.051, -40.847, 6.219, -32.356, -5.259]
  Call Extruder -0.38
  MoveL (T14089) to (103.84, 110.57, 15.7) mm, rotated rx 180 ry 0 rz -180 deg; joints [3.49, 72.949, -40.656, 6.512, -32.461, -5.501]
  Set speed (45.0 mm/s)
  Call Extruder -0.02
  MoveL (T14090) to (103.84, 110.57, 15.7) mm, rotated rx 180 ry 0 rz -180 deg; joints [3.49, 72.949, -40.656, 6.512, -32.461, -5.501]
  Set speed (150.0 mm/s)
  MoveL (T14091) to (103.84, 110.57, 17.7) mm, rotated rx 180 ry 0 rz -180 deg; joints [3.622, 72.609, -40.016, 6.702, -32.771, -5.643]
  MoveL (T14092) to (119.1, 110.71, 17.7) mm, rotated rx 180 ry 0 rz -180 deg; joints [3.622, 72.609, -40.016, 6.702, -32.771, -5.643]
  MoveL (T14093) to (119.1, 110.71, 15.7) mm, rotated rx 180 ry 0 rz -180 deg; joints [3.694, 72.008, -38.886, 6.738, -33.305, -5.64]
  Set speed (40.0 mm/s)
  Call Extruder 2.0
  MoveL (T14094) to (119.1, 110.71, 15.7) mm, rotated rx 180 ry 0 rz -180 deg; joints [3.694, 72.008, -38.886, 6.738, -33.305, -5.64]
  Set speed (26.8 mm/s)
  MoveL (T14095) to (119.1, 110.71, 15.7) mm, rotated rx 180 ry 0 rz -180 deg; joints [3.819, 66.837, -29.155, 6.233, -37.846, -4.929]
  Call Extruder 0.00302
  MoveL (T14096) to (119.1, 110.81, 15.7) mm, rotated rx 180 ry 0 rz -180 deg; joints [3.819, 66.837, -29.155, 6.233, -37.846, -4.929]
  Call Extruder 0.01378
  MoveL (T14097) to (119.42, 111.13, 15.7) mm, rotated rx 180 ry 0 rz -180 deg; joints [3.819, 66.837, -29.155, 6.233, -37.846, -4.929]
  Call Extruder 0.02805
  MoveL (T14098) to (120.34, 111.13, 15.7) mm, rotated rx 180 ry 0 rz -180 deg; joints [3.819, 66.837, -29.155, 6.233, -37.846, -4.929]
  Call Extruder 0.03515
  MoveL (T14099) to (121.16, 111.94, 15.7) mm, rotated rx 180 ry 0 rz -180 deg; joints [3.819, 66.837, -29.155, 6.233, -37.846, -4.929]
  Call Extruder 0.02988
  MoveL (T14100) to (121.16, 112.92, 15.7) mm, rotated rx 180 ry 0 rz -180 deg; joints [3.819, 66.837, -29.155, 6.233, -37.846, -4.929]
  Call Extruder 0.04453
  MoveL (T14101) to (119.69, 112.92, 15.7) mm, rotated rx 180 ry 0 rz -180 deg; joints [3.819, 66.837, -29.155, 6.233, -37.846, -4.929]
  Set speed (150.0 mm/s)
  MoveL (T14102) to (121, 113.15, 15.7) mm, rotated rx 180 ry 0 rz -180 deg; joints [3.819, 66.837, -29.155, 6.233, -37.846, -4.929]
  Set speed (26.8 mm/s)
  MoveL (T14103) to (121, 113.15, 15.7) mm, rotated rx 180 ry 0 rz -180 deg; joints [3.827, 66.561, -28.636, 6.211, -38.088, -4.896]
  Call Extruder 0.01587
  MoveL (T14104) to (120.65, 113.5, 15.7) mm, rotated rx 180 ry 0 rz -180 deg; joints [3.827, 66.561, -28.636, 6.211, -38.088, -4.896]
  Call Extruder 0.01955
  MoveL (T14105) to (120.04, 113.5, 15.7) mm, rotated rx 180 ry 0 rz -180 deg; joints [3.827, 66.561, -28.636, 6.211, -38.088, -4.896]
  Call Extruder 0.00755
  MoveL (T14106) to (120.21, 113.33, 15.7) mm, rotated rx 180 ry 0 rz -180 deg; joints [3.827, 66.561, -28.636, 6.211, -38.088, -4.896]
  Call Extruder 0.01955
  MoveL (T14107) to (119.6, 113.33, 15.7) mm, rotated rx 180 ry 0 rz -180 deg; joints [3.827, 66.561, -28.636, 6.211, -38.088, -4.896]
  Call Extruder 0.01276
  MoveL (T14108) to (119.32, 113.61, 15.7) mm, rotated rx 180 ry 0 rz -180 deg; joints [1.407, 66.288, -28.531, 2.298, -37.78, -1.816]
  Set speed (45.0 mm/s)
  Call Extruder -1.6
  MoveL (T14109) to (119.32, 113.61, 15.7) mm, rotated rx 180 ry 0 rz -180 deg; joints [1.407, 66.526, -28.571, 2.287, -37.977, -1.803]
  Set speed (120.0 mm/s)
  MoveL (T14110) to (119.32, 113.61, 15.7) mm, rotated rx 180 ry 0 rz -180 deg; joints [1.407, 66.526, -28.571, 2.287, -37.977, -1.803]
  Call Extruder -0.14126
  MoveL (T14111) to (119.6, 113.33, 15.7) mm, rotated rx 180 ry 0 rz -180 deg; joints [1.407, 66.526, -28.571, 2.287, -37.977, -1.803]
  Call Extruder -0.21639
  MoveL (T14112) to (120.21, 113.33, 15.7) mm, rotated rx 180 ry 0 rz -180 deg; joints [1.407, 66.526, -28.571, 2.287, -37.977, -1.803]
  Call Extruder -0.02235
  MoveL (T14113) to (120.17, 113.38, 15.7) mm, rotated rx 180 ry 0 rz -180 deg; joints [1.407, 66.526, -28.571, 2.287, -37.977, -1.803]
  Set speed (45.0 mm/s)
  Call Extruder -0.02
  MoveL (T14114) to (120.17, 113.38, 15.7) mm, rotated rx 180 ry 0 rz -180 deg; joints [1.407, 66.526, -28.571, 2.287, -37.977, -1.803]
  Set speed (150.0 mm/s)
  MoveL (T14115) to (120.17, 113.38, 17.7) mm, rotated rx 180 ry 0 rz -180 deg; joints [1.363, 71.364, -37.673, 2.456, -33.715, -2.044]
  MoveL (T14116) to (120.92, 110.35, 17.7) mm, rotated rx 180 ry 0 rz -180 deg; joints [1.363, 71.364, -37.673, 2.456, -33.715, -2.044]
  MoveL (T14117) to (120.92, 110.35, 15.7) mm, rotated rx 180 ry 0 rz -180 deg; joints [3.241, 71.591, -38.101, 5.86, -33.629, -4.884]
  Set speed (40.0 mm/s)
  Call Extruder 2.0
  MoveL (T14118) to (120.92, 110.35, 15.7) mm, rotated rx 180 ry 0 rz -180 deg; joints [3.351, 66.512, -28.544, 5.437, -38.093, -4.284]
  Set speed (26.8 mm/s)
  MoveL (T14119) to (120.92, 110.35, 15.7) mm, rotated rx 180 ry 0 rz -180 deg; joints [3.351, 66.512, -28.544, 5.437, -38.093, -4.284]
  Call Extruder 0.01747
  MoveL (T14120) to (120.55, 110.72, 15.7) mm, rotated rx 180 ry 0 rz -180 deg; joints [1.409, 66.321, -28.185, 2.282, -38.158, -1.794]
  Call Extruder 0.0208
  MoveL (T14121) to (119.92, 110.72, 15.7) mm, rotated rx 180 ry 0 rz -180 deg; joints [1.409, 66.321, -28.185, 2.282, -38.158, -1.794]
  Call Extruder 0.01747
  MoveL (T14122) to (120.3, 110.35, 15.7) mm, rotated rx 180 ry 0 rz -180 deg; joints [1.407, 66.511, -28.542, 2.287, -37.991, -1.803]
  Set speed (45.0 mm/s)
  Call Extruder -1.6
  MoveL (T14123) to (120.3, 110.35, 15.7) mm, rotated rx 180 ry 0 rz -180 deg; joints [1.407, 66.511, -28.542, 2.287, -37.991, -1.803]
  Set speed (120.0 mm/s)
  MoveL (T14124) to (120.3, 110.35, 15.7) mm, rotated rx 180 ry 0 rz -180 deg; joints [1.365, 66.317, -28.177, 2.21, -38.16, -1.738]
  Call Extruder -0.18758
  MoveL (T14125) to (119.92, 110.72, 15.7) mm, rotated rx 180 ry 0 rz -180 deg; joints [1.365, 66.317, -28.177, 2.21, -38.16, -1.738]
  Call Extruder -0.19242
  MoveL (T14126) to (120.46, 110.72, 15.7) mm, rotated rx 180 ry 0 rz -180 deg; joints [1.365, 66.317, -28.177, 2.21, -38.16, -1.738]
  Set speed (45.0 mm/s)
  Call Extruder -0.02
  MoveL (T14127) to (120.46, 110.72, 15.7) mm, rotated rx 180 ry 0 rz -180 deg; joints [1.365, 66.317, -28.177, 2.21, -38.16, -1.738]
  Set speed (150.0 mm/s)
  MoveL (T14128) to (120.46, 110.72, 17.7) mm, rotated rx 180 ry 0 rz -180 deg; joints [1.365, 66.317, -28.177, 2.21, -38.16, -1.738]
  MoveL (T14129) to (104.34, 103.54, 17.7) mm, rotated rx 180 ry 0 rz -180 deg; joints [1.365, 66.317, -28.177, 2.21, -38.16, -1.738]
  MoveL (T14130) to (104.34, 103.54, 15.9) mm, rotated rx 180 ry 0 rz -180 deg; joints [1.319, 71.489, -37.909, 2.385, -33.603, -1.986]
  Set speed (40.0 mm/s)
  Call Extruder 2.0
  MoveL (T14131) to (104.34, 103.54, 15.9) mm, rotated rx 180 ry 0 rz -180 deg; joints [1.319, 71.489, -37.909, 2.385, -33.603, -1.986]
  Set speed (26.8 mm/s)
  MoveL (T14132) to (104.34, 103.54, 15.9) mm, rotated rx 180 ry 0 rz -180 deg; joints [3.282, 71.728, -38.358, 5.951, -33.512, -4.967]
  Call Extruder 0.07565
  MoveL (T14133) to (106.82, 103.54, 15.9) mm, rotated rx 180 ry 0 rz -180 deg; joints [3.398, 66.414, -28.36, 5.502, -38.183, -4.33]
  Call Extruder 0.05793
  MoveL (T14134) to (106.82, 105.44, 15.9) mm, rotated rx 180 ry 0 rz -180 deg; joints [3.398, 66.414, -28.36, 5.502, -38.183, -4.33]
  Call Extruder 0.11362
  MoveL (T14135) to (110.55, 105.44, 15.9) mm, rotated rx 180 ry 0 rz -180 deg; joints [3.398, 66.414, -28.36, 5.502, -38.183, -4.33]
  Call Extruder 0.05793
  MoveL (T14136) to (110.55, 103.54, 15.9) mm, rotated rx 180 ry 0 rz -180 deg; joints [1.366, 66.215, -27.985, 2.207, -38.25, -1.734]
  Call Extruder 0.09938
  MoveL (T14137) to (113.81, 103.54, 15.9) mm, rotated rx 180 ry 0 rz -180 deg; joints [1.366, 66.215, -27.985, 2.207, -38.25, -1.734]
  Call Extruder 0.05793
  MoveL (T14138) to (113.81, 105.44, 15.9) mm, rotated rx 180 ry 0 rz -180 deg; joints [1.365, 66.301, -28.148, 2.21, -38.174, -1.737]
  Call Extruder 0.11352
  MoveL (T14139) to (117.54, 105.44, 15.9) mm, rotated rx 180 ry 0 rz -180 deg; joints [1.365, 66.301, -28.148, 2.21, -38.174, -1.737]
  Call Extruder 0.05793
  MoveL (T14140) to (117.54, 103.54, 15.9) mm, rotated rx 180 ry 0 rz -180 deg; joints [1.365, 66.301, -28.148, 2.21, -38.174, -1.737]
  Call Extruder 0.11943
  MoveL (T14141) to (121.46, 103.54, 15.9) mm, rotated rx 180 ry 0 rz -180 deg; joints [1.365, 66.301, -28.148, 2.21, -38.174, -1.737]
  Call Extruder 0.08385
  MoveL (T14142) to (121.46, 106.29, 15.9) mm, rotated rx 180 ry 0 rz -180 deg; joints [1.332, 66.109, -27.787, 2.148, -38.342, -1.685]
  Call Extruder 0.05863
  MoveL (T14143) to (119.54, 106.29, 15.9) mm, rotated rx 180 ry 0 rz -180 deg; joints [1.332, 66.109, -27.787, 2.148, -38.342, -1.685]
  Call Extruder 0.11631
  MoveL (T14144) to (119.53, 110.11, 15.9) mm, rotated rx 180 ry 0 rz -180 deg; joints [1.332, 66.109, -27.787, 2.148, -38.342, -1.685]
  Call Extruder 0.05868
  MoveL (T14145) to (121.46, 110.11, 15.9) mm, rotated rx 180 ry 0 rz -180 deg; joints [1.332, 66.109, -27.787, 2.148, -38.342, -1.685]
  Call Extruder 0.11593
  MoveL (T14146) to (121.46, 113.92, 15.9) mm, rotated rx 180 ry 0 rz -180 deg; joints [1.332, 66.109, -27.787, 2.148, -38.342, -1.685]
  Call Extruder 0.05873
  MoveL (T14147) to (119.53, 113.91, 15.9) mm, rotated rx 180 ry 0 rz -180 deg; joints [1.323, 66.109, -27.786, 2.133, -38.342, -1.673]
  Call Extruder 0.11564
  MoveL (T14148) to (119.53, 117.71, 15.9) mm, rotated rx 180 ry 0 rz -180 deg; joints [1.276, 71.615, -38.145, 2.313, -33.491, -1.929]
  Call Extruder 0.05879
  MoveL (T14149) to (121.46, 117.71, 15.9) mm, rotated rx 180 ry 0 rz -180 deg; joints [3.322, 71.865, -38.617, 6.043, -33.395, -5.051]
  Call Extruder 0.11423
  MoveL (T14150) to (121.46, 121.46, 15.9) mm, rotated rx 180 ry 0 rz -180 deg; joints [3.322, 71.865, -38.617, 6.043, -33.395, -5.051]
  Call Extruder 0.54596
  MoveL (T14151) to (103.54, 121.46, 15.9) mm, rotated rx 180 ry 0 rz -180 deg; joints [3.445, 66.316, -28.176, 5.566, -38.272, -4.375]
  Call Extruder 0.54596
  MoveL (T14152) to (103.54, 103.54, 15.9) mm, rotated rx 180 ry 0 rz -180 deg; joints [3.445, 66.316, -28.176, 5.566, -38.272, -4.375]
  Call Extruder 0.02254
  MoveL (T14153) to (104.28, 103.54, 15.9) mm, rotated rx 180 ry 0 rz -180 deg; joints [3.445, 66.316, -28.176, 5.566, -38.272, -4.375]
  Set speed (150.0 mm/s)
  MoveL (T14154) to (103.53, 103.13, 15.9) mm, rotated rx 180 ry 0 rz -180 deg; joints [1.339, 66.11, -27.788, 2.159, -38.342, -1.693]
  Set speed (26.8 mm/s)
  MoveL (T14155) to (103.53, 103.13, 15.9) mm, rotated rx 180 ry 0 rz -180 deg; joints [1.339, 66.11, -27.788, 2.159, -38.342, -1.693]
  Call Extruder 0.11264
  MoveL (T14156) to (107.23, 103.13, 15.9) mm, rotated rx 180 ry 0 rz -180 deg; joints [1.339, 66.11, -27.788, 2.159, -38.342, -1.693]
  Call Extruder 0.05793
  MoveL (T14157) to (107.23, 105.03, 15.9) mm, rotated rx 180 ry 0 rz -180 deg; joints [1.326, 66.124, -27.815, 2.138, -38.328, -1.678]
  Call Extruder 0.08882
  MoveL (T14158) to (110.14, 105.03, 15.9) mm, rotated rx 180 ry 0 rz -180 deg; joints [1.326, 66.124, -27.815, 2.138, -38.328, -1.678]
  Call Extruder 0.05793
  MoveL (T14159) to (110.14, 103.13, 15.9) mm, rotated rx 180 ry 0 rz -180 deg; joints [1.326, 66.124, -27.815, 2.138, -38.328, -1.678]
  Call Extruder 0.12417
  MoveL (T14160) to (114.22, 103.13, 15.9) mm, rotated rx 180 ry 0 rz -180 deg; joints [1.326, 66.124, -27.815, 2.138, -38.328, -1.678]
  Call Extruder 0.05793
  MoveL (T14161) to (114.22, 105.03, 15.9) mm, rotated rx 180 ry 0 rz -180 deg; joints [1.326, 66.124, -27.815, 2.138, -38.328, -1.678]
  Call Extruder 0.08871
  MoveL (T14162) to (117.13, 105.03, 15.9) mm, rotated rx 180 ry 0 rz -180 deg; joints [1.326, 66.124, -27.815, 2.138, -38.328, -1.678]
  Call Extruder 0.05793
  MoveL (T14163) to (117.13, 103.13, 15.9) mm, rotated rx 180 ry 0 rz -180 deg; joints [1.326, 66.124, -27.815, 2.138, -38.328, -1.678]
  Call Extruder 0.14424
  MoveL (T14164) to (121.87, 103.13, 15.9) mm, rotated rx 180 ry 0 rz -180 deg; joints [1.326, 66.124, -27.815, 2.138, -38.328, -1.678]
  Call Extruder 0.10865
  MoveL (T14165) to (121.87, 106.7, 15.9) mm, rotated rx 180 ry 0 rz -180 deg; joints [1.326, 66.124, -27.815, 2.138, -38.328, -1.678]
  Call Extruder 0.05864
  MoveL (T14166) to (119.94, 106.7, 15.9) mm, rotated rx 180 ry 0 rz -180 deg; joints [1.326, 66.124, -27.815, 2.138, -38.328, -1.678]
  Call Extruder 0.09151
  MoveL (T14167) to (119.94, 109.7, 15.9) mm, rotated rx 180 ry 0 rz -180 deg; joints [1.323, 66.109, -27.786, 2.133, -38.342, -1.673]
  Call Extruder 0.05868
  MoveL (T14168) to (121.87, 109.7, 15.9) mm, rotated rx 180 ry 0 rz -180 deg; joints [1.321, 66.344, -28.228, 2.139, -38.135, -1.683]
  Call Extruder 0.14076
  MoveL (T14169) to (121.87, 114.32, 15.9) mm, rotated rx 180 ry 0 rz -180 deg; joints [1.321, 66.344, -28.228, 2.139, -38.135, -1.683]
  Call Extruder 0.05874
  MoveL (T14170) to (119.94, 114.32, 15.9) mm, rotated rx 180 ry 0 rz -180 deg; joints [1.321, 66.344, -28.228, 2.139, -38.135, -1.683]
  Call Extruder 0.09084
  MoveL (T14171) to (119.94, 117.3, 15.9) mm, rotated rx 180 ry 0 rz -180 deg; joints [1.321, 66.344, -28.228, 2.139, -38.135, -1.683]
  Call Extruder 0.05878
  MoveL (T14172) to (121.87, 117.31, 15.9) mm, rotated rx 180 ry 0 rz -180 deg; joints [1.321, 66.344, -28.228, 2.139, -38.135, -1.683]
  Call Extruder 0.13901
  MoveL (T14173) to (121.87, 121.87, 15.9) mm, rotated rx 180 ry 0 rz -180 deg; joints [1.321, 66.344, -28.228, 2.139, -38.135, -1.683]
  Call Extruder 0.57077
  MoveL (T14174) to (103.13, 121.87, 15.9) mm, rotated rx 180 ry 0 rz -180 deg; joints [1.321, 66.344, -28.228, 2.139, -38.135, -1.683]
  Call Extruder 0.57077
  MoveL (T14175) to (103.13, 103.13, 15.9) mm, rotated rx 180 ry 0 rz -180 deg; joints [1.321, 66.105, -28.188, 2.149, -37.937, -1.695]
  Call Extruder 0.01036
  MoveL (T14176) to (103.47, 103.13, 15.9) mm, rotated rx 180 ry 0 rz -180 deg; joints [3.142, 71.301, -37.949, 5.702, -33.483, -4.761]
  Set speed (150.0 mm/s)
  MoveL (T14177) to (102.72, 102.81, 15.9) mm, rotated rx 180 ry 0 rz -180 deg; joints [3.142, 71.536, -37.997, 5.674, -33.669, -4.727]
  Set speed (25.0 mm/s)
  MoveL (T14178) to (102.72, 102.81, 15.9) mm, rotated rx 180 ry 0 rz -180 deg; joints [3.142, 71.536, -37.997, 5.674, -33.669, -4.727]
  Call Extruder 0.00259
  MoveL (T14179) to (102.72, 102.72, 15.9) mm, rotated rx 180 ry 0 rz -180 deg; joints [3.142, 71.536, -37.997, 5.674, -33.669, -4.727]
  Call Extruder 0.14964
  MoveL (T14180) to (107.64, 102.72, 15.9) mm, rotated rx 180 ry 0 rz -180 deg; joints [3.142, 71.536, -37.997, 5.674, -33.669, -4.727]
  Call Extruder 0.05793
  MoveL (T14181) to (107.64, 104.63, 15.9) mm, rotated rx 180 ry 0 rz -180 deg; joints [3.142, 71.536, -37.997, 5.674, -33.669, -4.727]
  Call Extruder 0.06401
  MoveL (T14182) to (109.74, 104.63, 15.9) mm, rotated rx 180 ry 0 rz -180 deg; joints [3.142, 71.536, -37.997, 5.674, -33.669, -4.727]
  Call Extruder 0.05793
  MoveL (T14183) to (109.74, 102.72, 15.9) mm, rotated rx 180 ry 0 rz -180 deg; joints [3.142, 71.536, -37.997, 5.674, -33.669, -4.727]
  Call Extruder 0.14896
  MoveL (T14184) to (114.63, 102.72, 15.9) mm, rotated rx 180 ry 0 rz -180 deg; joints [3.142, 71.536, -37.997, 5.674, -33.669, -4.727]
  Call Extruder 0.05793
  MoveL (T14185) to (114.63, 104.63, 15.9) mm, rotated rx 180 ry 0 rz -180 deg; joints [3.142, 71.536, -37.997, 5.674, -33.669, -4.727]
  Call Extruder 0.06391
  MoveL (T14186) to (116.73, 104.63, 15.9) mm, rotated rx 180 ry 0 rz -180 deg; joints [3.214, 71.343, -37.635, 5.778, -33.844, -4.804]
  Call Extruder 0.05793
  MoveL (T14187) to (116.73, 102.72, 15.9) mm, rotated rx 180 ry 0 rz -180 deg; joints [3.214, 71.343, -37.635, 5.778, -33.844, -4.804]
  Call Extruder 0.16905
  MoveL (T14188) to (122.28, 102.72, 15.9) mm, rotated rx 180 ry 0 rz -180 deg; joints [3.214, 71.343, -37.635, 5.778, -33.844, -4.804]
  Call Extruder 0.13344
  MoveL (T14189) to (122.28, 107.11, 15.9) mm, rotated rx 180 ry 0 rz -180 deg; joints [3.214, 71.343, -37.635, 5.778, -33.844, -4.804]
  Call Extruder 0.05864
  MoveL (T14190) to (120.35, 107.11, 15.9) mm, rotated rx 180 ry 0 rz -180 deg; joints [3.217, 71.162, -37.294, 5.76, -34.003, -4.78]
  Call Extruder 0.06671
  MoveL (T14191) to (120.35, 109.3, 15.9) mm, rotated rx 180 ry 0 rz -180 deg; joints [3.217, 71.162, -37.294, 5.76, -34.003, -4.78]
  Call Extruder 0.05867
  MoveL (T14192) to (122.28, 109.3, 15.9) mm, rotated rx 180 ry 0 rz -180 deg; joints [3.217, 71.162, -37.294, 5.76, -34.003, -4.78]
  Call Extruder 0.16558
  MoveL (T14193) to (122.28, 114.73, 15.9) mm, rotated rx 180 ry 0 rz -180 deg; joints [3.102, 71.471, -37.875, 5.593, -33.722, -4.657]
  Call Extruder 0.05875
  MoveL (T14194) to (120.35, 114.73, 15.9) mm, rotated rx 180 ry 0 rz -180 deg; joints [3.041, 71.461, -37.857, 5.483, -33.726, -4.564]
  Call Extruder 0.06604
  MoveL (T14195) to (120.35, 116.9, 15.9) mm, rotated rx 180 ry 0 rz -180 deg; joints [3.041, 71.461, -37.857, 5.483, -33.726, -4.564]
  Call Extruder 0.05877
  MoveL (T14196) to (122.28, 116.9, 15.9) mm, rotated rx 180 ry 0 rz -180 deg; joints [3.041, 71.461, -37.857, 5.483, -33.726, -4.564]
  Call Extruder 0.1638
  MoveL (T14197) to (122.28, 122.28, 15.9) mm, rotated rx 180 ry 0 rz -180 deg; joints [3.221, 70.983, -36.956, 5.743, -34.161, -4.757]
  Call Extruder 0.59557
  MoveL (T14198) to (102.72, 122.28, 15.9) mm, rotated rx 180 ry 0 rz -180 deg; joints [3.221, 70.983, -36.956, 5.743, -34.161, -4.757]
  Call Extruder 0.59115
  MoveL (T14199) to (102.72, 102.87, 15.9) mm, rotated rx 180 ry 0 rz -180 deg; joints [3.221, 70.983, -36.956, 5.743, -34.161, -4.757]
  Set speed (150.0 mm/s)
  MoveL (T14200) to (102.78, 102.75, 15.9) mm, rotated rx 180 ry 0 rz -180 deg; joints [3.224, 70.805, -36.621, 5.726, -34.317, -4.734]
  Set speed (45.0 mm/s)
  Call Extruder -1.6
  MoveL (T14201) to (102.78, 102.75, 15.9) mm, rotated rx 180 ry 0 rz -180 deg; joints [3.224, 70.805, -36.621, 5.726, -34.317, -4.734]
  Set speed (120.0 mm/s)
  MoveL (T14202) to (102.78, 102.75, 15.9) mm, rotated rx 180 ry 0 rz -180 deg; joints [2.98, 71.452, -37.839, 5.372, -33.73, -4.472]
  Call Extruder -0.05166
  MoveL (T14203) to (102.72, 102.72, 15.9) mm, rotated rx 180 ry 0 rz -180 deg; joints [2.98, 71.452, -37.839, 5.372, -33.73, -4.472]
  Call Extruder -0.32834
  MoveL (T14204) to (103.65, 102.72, 15.9) mm, rotated rx 180 ry 0 rz -180 deg; joints [2.919, 71.442, -37.821, 5.262, -33.733, -4.38]
  Set speed (45.0 mm/s)
  Call Extruder -0.02
  MoveL (T14205) to (103.65, 102.72, 15.9) mm, rotated rx 180 ry 0 rz -180 deg; joints [2.919, 71.442, -37.821, 5.262, -33.733, -4.38]
  Set speed (150.0 mm/s)
  MoveL (T14206) to (103.65, 102.72, 17.9) mm, rotated rx 180 ry 0 rz -180 deg; joints [2.919, 71.442, -37.821, 5.262, -33.733, -4.38]
  MoveL (T14207) to (106.29, 103.84, 17.9) mm, rotated rx 180 ry 0 rz -180 deg; joints [3.228, 70.628, -36.288, 5.709, -34.473, -4.711]
  MoveL (T14208) to (106.29, 103.84, 15.9) mm, rotated rx 180 ry 0 rz -180 deg; joints [3.228, 70.628, -36.288, 5.709, -34.473, -4.711]
  Set speed (40.0 mm/s)
  Call Extruder 2.0
  MoveL (T14209) to (106.29, 103.84, 15.9) mm, rotated rx 180 ry 0 rz -180 deg; joints [3.231, 70.453, -35.959, 5.693, -34.627, -4.689]
  Set speed (26.8 mm/s)
  MoveL (T14210) to (106.29, 103.84, 15.9) mm, rotated rx 180 ry 0 rz -180 deg; joints [3.231, 70.453, -35.959, 5.693, -34.627, -4.689]
  Call Extruder 0.07441
  MoveL (T14211) to (103.84, 103.84, 15.9) mm, rotated rx 180 ry 0 rz -180 deg; joints [2.858, 71.433, -37.804, 5.152, -33.737, -4.288]
  Call Extruder 0.7458
  MoveL (T14212) to (121.16, 121.16, 15.9) mm, rotated rx 180 ry 0 rz -180 deg; joints [2.858, 71.433, -37.804, 5.152, -33.737, -4.288]
  Call Extruder 0.09564
  MoveL (T14213) to (121.16, 118.02, 15.9) mm, rotated rx 180 ry 0 rz -180 deg; joints [2.797, 71.424, -37.787, 5.041, -33.74, -4.195]
  Call Extruder 0.0108
  MoveL (T14214) to (120.8, 118.02, 15.9) mm, rotated rx 180 ry 0 rz -180 deg; joints [2.797, 71.424, -37.787, 5.041, -33.74, -4.195]
  Call Extruder 0.13527
  MoveL (T14215) to (117.66, 121.16, 15.9) mm, rotated rx 180 ry 0 rz -180 deg; joints [3.235, 70.279, -35.631, 5.677, -34.779, -4.668]
  Call Extruder 0.03385
  MoveL (T14216) to (116.55, 121.16, 15.9) mm, rotated rx 180 ry 0 rz -180 deg; joints [3.235, 70.279, -35.631, 5.677, -34.779, -4.668]
  Call Extruder 0.54738
  MoveL (T14217) to (103.84, 108.45, 15.9) mm, rotated rx 180 ry 0 rz -180 deg; joints [3.238, 70.106, -35.306, 5.661, -34.931, -4.646]
  Call Extruder 0.03385
  MoveL (T14218) to (103.84, 107.34, 15.9) mm, rotated rx 180 ry 0 rz -180 deg; joints [3.238, 70.106, -35.306, 5.661, -34.931, -4.646]
  Call Extruder 0.11512
  MoveL (T14219) to (106.52, 104.67, 15.9) mm, rotated rx 180 ry 0 rz -180 deg; joints [3.238, 70.106, -35.306, 5.661, -34.931, -4.646]
  Call Extruder 0.03288
  MoveL (T14220) to (106.52, 105.75, 15.9) mm, rotated rx 180 ry 0 rz -180 deg; joints [2.737, 71.415, -37.77, 4.931, -33.744, -4.103]
  Call Extruder 0.04153
  MoveL (T14221) to (107.88, 105.75, 15.9) mm, rotated rx 180 ry 0 rz -180 deg; joints [2.737, 71.415, -37.77, 4.931, -33.744, -4.103]
  Set speed (45.0 mm/s)
  Call Extruder -1.6
  MoveL (T14222) to (107.88, 105.75, 15.9) mm, rotated rx 180 ry 0 rz -180 deg; joints [2.676, 71.407, -37.754, 4.82, -33.747, -4.011]
  Set speed (120.0 mm/s)
  MoveL (T14223) to (107.88, 105.75, 15.9) mm, rotated rx 180 ry 0 rz -180 deg; joints [2.676, 71.407, -37.754, 4.82, -33.747, -4.011]
  Call Extruder -0.38
  MoveL (T14224) to (106.81, 105.75, 15.9) mm, rotated rx 180 ry 0 rz -180 deg; joints [3.242, 69.935, -34.984, 5.646, -35.082, -4.625]
  Set speed (45.0 mm/s)
  Call Extruder -0.02
  MoveL (T14225) to (106.81, 105.75, 15.9) mm, rotated rx 180 ry 0 rz -180 deg; joints [3.242, 69.935, -34.984, 5.646, -35.082, -4.625]
  Set speed (150.0 mm/s)
  MoveL (T14226) to (106.81, 105.75, 17.9) mm, rotated rx 180 ry 0 rz -180 deg; joints [3.242, 69.935, -34.984, 5.646, -35.082, -4.625]
  MoveL (T14227) to (110.54, 105.78, 17.9) mm, rotated rx 180 ry 0 rz -180 deg; joints [3.245, 69.765, -34.664, 5.631, -35.232, -4.605]
  MoveL (T14228) to (110.54, 105.78, 15.9) mm, rotated rx 180 ry 0 rz -180 deg; joints [3.245, 69.765, -34.664, 5.631, -35.232, -4.605]
  Set speed (40.0 mm/s)
  Call Extruder 2.0
  MoveL (T14229) to (110.54, 105.78, 15.9) mm, rotated rx 180 ry 0 rz -180 deg; joints [2.615, 71.398, -37.738, 4.71, -33.75, -3.919]
  Set speed (26.8 mm/s)
  MoveL (T14230) to (110.54, 105.78, 15.9) mm, rotated rx 180 ry 0 rz -180 deg; joints [2.615, 71.398, -37.738, 4.71, -33.75, -3.919]
  Call Extruder 0.00424
  MoveL (T14231) to (110.64, 105.87, 15.9) mm, rotated rx 180 ry 0 rz -180 deg; joints [2.615, 71.398, -37.738, 4.71, -33.75, -3.919]
  Call Extruder 0.01452
  MoveL (T14232) to (111.12, 105.87, 15.9) mm, rotated rx 180 ry 0 rz -180 deg; joints [2.615, 71.398, -37.738, 4.71, -33.75, -3.919]
  Call Extruder 0.01375
  MoveL (T14233) to (111.44, 105.55, 15.9) mm, rotated rx 180 ry 0 rz -180 deg; joints [2.554, 71.39, -37.722, 4.6, -33.753, -3.827]
  Call Extruder 0.03663
  MoveL (T14234) to (111.44, 104.35, 15.9) mm, rotated rx 180 ry 0 rz -180 deg; joints [2.554, 71.39, -37.722, 4.6, -33.753, -3.827]
  Call Extruder 0.02185
  MoveL (T14235) to (111.94, 103.84, 15.9) mm, rotated rx 180 ry 0 rz -180 deg; joints [2.554, 71.39, -37.722, 4.6, -33.753, -3.827]
  Call Extruder 0.02837
  MoveL (T14236) to (112.88, 103.84, 15.9) mm, rotated rx 180 ry 0 rz -180 deg; joints [3.249, 69.596, -34.346, 5.617, -35.38, -4.584]
  Call Extruder 0.04603
  MoveL (T14237) to (112.88, 105.36, 15.9) mm, rotated rx 180 ry 0 rz -180 deg; joints [3.249, 69.596, -34.346, 5.617, -35.38, -4.584]
  Set speed (150.0 mm/s)
  MoveL (T14238) to (113.1, 103.95, 15.9) mm, rotated rx 180 ry 0 rz -180 deg; joints [3.249, 69.596, -34.346, 5.617, -35.38, -4.584]
  Set speed (26.8 mm/s)
  MoveL (T14239) to (113.1, 103.95, 15.9) mm, rotated rx 180 ry 0 rz -180 deg; joints [3.252, 69.428, -34.03, 5.602, -35.528, -4.564]
  Call Extruder 0.01886
  MoveL (T14240) to (113.51, 104.36, 15.9) mm, rotated rx 180 ry 0 rz -180 deg; joints [3.252, 69.428, -34.03, 5.602, -35.528, -4.564]
  Call Extruder 0.02005
  MoveL (T14241) to (113.51, 104.98, 15.9) mm, rotated rx 180 ry 0 rz -180 deg; joints [2.493, 71.382, -37.707, 4.49, -33.756, -3.735]
  Call Extruder 0.01042
  MoveL (T14242) to (113.28, 104.75, 15.9) mm, rotated rx 180 ry 0 rz -180 deg; joints [2.493, 71.382, -37.707, 4.49, -33.756, -3.735]
  Call Extruder 0.02005
  MoveL (T14243) to (113.28, 105.37, 15.9) mm, rotated rx 180 ry 0 rz -180 deg; joints [2.493, 71.382, -37.707, 4.49, -33.756, -3.735]
  Call Extruder 0.01308
  MoveL (T14244) to (113.57, 105.65, 15.9) mm, rotated rx 180 ry 0 rz -180 deg; joints [2.493, 71.382, -37.707, 4.49, -33.756, -3.735]
  Set speed (45.0 mm/s)
  Call Extruder -1.6
  MoveL (T14245) to (113.57, 105.65, 15.9) mm, rotated rx 180 ry 0 rz -180 deg; joints [2.432, 71.374, -37.693, 4.38, -33.759, -3.643]
  Set speed (120.0 mm/s)
  MoveL (T14246) to (113.57, 105.65, 15.9) mm, rotated rx 180 ry 0 rz -180 deg; joints [2.432, 71.374, -37.693, 4.38, -33.759, -3.643]
  Call Extruder -0.14307
  MoveL (T14247) to (113.28, 105.37, 15.9) mm, rotated rx 180 ry 0 rz -180 deg; joints [3.256, 69.261, -33.716, 5.588, -35.674, -4.545]
  Call Extruder -0.21934
  MoveL (T14248) to (113.28, 104.75, 15.9) mm, rotated rx 180 ry 0 rz -180 deg; joints [3.256, 69.261, -33.716, 5.588, -35.674, -4.545]
  Call Extruder -0.01759
  MoveL (T14249) to (113.32, 104.78, 15.9) mm, rotated rx 180 ry 0 rz -180 deg; joints [3.256, 69.261, -33.716, 5.588, -35.674, -4.545]
  Set speed (45.0 mm/s)
  Call Extruder -0.02
  MoveL (T14250) to (113.32, 104.78, 15.9) mm, rotated rx 180 ry 0 rz -180 deg; joints [3.259, 69.096, -33.405, 5.575, -35.82, -4.525]
  Set speed (150.0 mm/s)
  MoveL (T14251) to (113.32, 104.78, 17.9) mm, rotated rx 180 ry 0 rz -180 deg; joints [3.259, 69.096, -33.405, 5.575, -35.82, -4.525]
  MoveL (T14252) to (110.67, 104.08, 17.9) mm, rotated rx 180 ry 0 rz -180 deg; joints [2.371, 71.367, -37.678, 4.269, -33.762, -3.551]
  MoveL (T14253) to (110.67, 104.08, 15.9) mm, rotated rx 180 ry 0 rz -180 deg; joints [2.371, 71.367, -37.678, 4.269, -33.762, -3.551]
  Set speed (40.0 mm/s)
  Call Extruder 2.0
  MoveL (T14254) to (110.67, 104.08, 15.9) mm, rotated rx 180 ry 0 rz -180 deg; joints [2.371, 71.367, -37.678, 4.269, -33.762, -3.551]
  Set speed (26.8 mm/s)
  MoveL (T14255) to (110.67, 104.08, 15.9) mm, rotated rx 180 ry 0 rz -180 deg; joints [2.31, 71.359, -37.664, 4.159, -33.765, -3.46]
  Call Extruder 0.01643
  MoveL (T14256) to (111.03, 104.43, 15.9) mm, rotated rx 180 ry 0 rz -180 deg; joints [2.31, 71.359, -37.664, 4.159, -33.765, -3.46]
  Call Extruder 0.0201
  MoveL (T14257) to (111.03, 105.05, 15.9) mm, rotated rx 180 ry 0 rz -180 deg; joints [3.263, 68.932, -33.096, 5.561, -35.964, -4.506]
  Call Extruder 0.01643
  MoveL (T14258) to (110.67, 104.69, 15.9) mm, rotated rx 180 ry 0 rz -180 deg; joints [3.263, 68.932, -33.096, 5.561, -35.964, -4.506]
  Set speed (45.0 mm/s)
  Call Extruder -1.6
  MoveL (T14259) to (110.67, 104.69, 15.9) mm, rotated rx 180 ry 0 rz -180 deg; joints [3.263, 68.932, -33.096, 5.561, -35.964, -4.506]
  Set speed (120.0 mm/s)
  MoveL (T14260) to (110.67, 104.69, 15.9) mm, rotated rx 180 ry 0 rz -180 deg; joints [3.266, 68.768, -32.789, 5.548, -36.108, -4.487]
  Call Extruder -0.17945
  MoveL (T14261) to (111.03, 105.05, 15.9) mm, rotated rx 180 ry 0 rz -180 deg; joints [3.266, 68.768, -32.789, 5.548, -36.108, -4.487]
  Call Extruder -0.20055
  MoveL (T14262) to (111.03, 104.49, 15.9) mm, rotated rx 180 ry 0 rz -180 deg; joints [3.266, 68.768, -32.789, 5.548, -36.108, -4.487]
  Set speed (45.0 mm/s)
  Call Extruder -0.02
  MoveL (T14263) to (111.03, 104.49, 15.9) mm, rotated rx 180 ry 0 rz -180 deg; joints [2.249, 71.352, -37.65, 4.049, -33.768, -3.368]
  Set speed (150.0 mm/s)
  MoveL (T14264) to (111.03, 104.49, 17.9) mm, rotated rx 180 ry 0 rz -180 deg; joints [2.249, 71.352, -37.65, 4.049, -33.768, -3.368]
  MoveL (T14265) to (117.12, 105.75, 17.9) mm, rotated rx 180 ry 0 rz -180 deg; joints [2.249, 71.352, -37.65, 4.049, -33.768, -3.368]
  MoveL (T14266) to (117.12, 105.75, 15.9) mm, rotated rx 180 ry 0 rz -180 deg; joints [2.188, 71.345, -37.637, 3.939, -33.77, -3.276]
  Set speed (40.0 mm/s)
  Call Extruder 2.0
  MoveL (T14267) to (117.12, 105.75, 15.9) mm, rotated rx 180 ry 0 rz -180 deg; joints [2.188, 71.345, -37.637, 3.939, -33.77, -3.276]
  Set speed (26.8 mm/s)
  MoveL (T14268) to (117.12, 105.75, 15.9) mm, rotated rx 180 ry 0 rz -180 deg; joints [3.27, 68.606, -32.484, 5.535, -36.25, -4.469]
  Call Extruder 0.02211
  MoveL (T14269) to (117.85, 105.75, 15.9) mm, rotated rx 180 ry 0 rz -180 deg; joints [3.27, 68.606, -32.484, 5.535, -36.25, -4.469]
  Call Extruder 0.0523
  MoveL (T14270) to (117.85, 104.03, 15.9) mm, rotated rx 180 ry 0 rz -180 deg; joints [3.273, 68.445, -32.18, 5.522, -36.392, -4.45]
  Call Extruder 0.08435
  MoveL (T14271) to (119.8, 105.99, 15.9) mm, rotated rx 180 ry 0 rz -180 deg; joints [3.273, 68.445, -32.18, 5.522, -36.392, -4.45]
  Call Extruder 0.04118
  MoveL (T14272) to (121.16, 105.99, 15.9) mm, rotated rx 180 ry 0 rz -180 deg; joints [2.127, 71.338, -37.624, 3.829, -33.773, -3.184]
  Call Extruder 0.06525
  MoveL (T14273) to (121.16, 103.84, 15.9) mm, rotated rx 180 ry 0 rz -180 deg; joints [2.127, 71.338, -37.624, 3.829, -33.773, -3.184]
  Call Extruder 0.7458
  MoveL (T14274) to (103.84, 121.16, 15.9) mm, rotated rx 180 ry 0 rz -180 deg; joints [2.127, 71.338, -37.624, 3.829, -33.773, -3.184]
  Call Extruder 0.10645
  MoveL (T14275) to (103.84, 117.66, 15.9) mm, rotated rx 180 ry 0 rz -180 deg; joints [2.067, 71.331, -37.612, 3.719, -33.775, -3.093]
  Call Extruder 0.15054
  MoveL (T14276) to (107.34, 121.16, 15.9) mm, rotated rx 180 ry 0 rz -180 deg; joints [2.067, 71.331, -37.612, 3.719, -33.775, -3.093]
  Call Extruder 0.03385
  MoveL (T14277) to (108.45, 121.16, 15.9) mm, rotated rx 180 ry 0 rz -180 deg; joints [3.277, 68.285, -31.88, 5.51, -36.532, -4.432]
  Call Extruder 0.45881
  MoveL (T14278) to (119.1, 110.51, 15.9) mm, rotated rx 180 ry 0 rz -180 deg; joints [3.277, 68.285, -31.88, 5.51, -36.532, -4.432]
  Call Extruder 0.00933
  MoveL (T14279) to (119.1, 110.2, 15.9) mm, rotated rx 180 ry 0 rz -180 deg; joints [3.277, 68.285, -31.88, 5.51, -36.532, -4.432]
  Call Extruder 0.00558
  MoveL (T14280) to (119.23, 110.07, 15.9) mm, rotated rx 180 ry 0 rz -180 deg; joints [3.28, 68.126, -31.58, 5.498, -36.672, -4.414]
  Call Extruder 0.00159
  MoveL (T14281) to (119.23, 110.02, 15.9) mm, rotated rx 180 ry 0 rz -180 deg; joints [3.28, 68.126, -31.58, 5.498, -36.672, -4.414]
  Call Extruder 0.18406
  MoveL (T14282) to (114.96, 105.75, 15.9) mm, rotated rx 180 ry 0 rz -180 deg; joints [2.006, 71.325, -37.6, 3.609, -33.778, -3.001]
  Call Extruder 0.0094
  MoveL (T14283) to (114.65, 105.75, 15.9) mm, rotated rx 180 ry 0 rz -180 deg; joints [2.006, 71.325, -37.6, 3.609, -33.778, -3.001]
  Call Extruder 0.46547
  MoveL (T14284) to (103.84, 116.55, 15.9) mm, rotated rx 180 ry 0 rz -180 deg; joints [1.945, 71.319, -37.588, 3.499, -33.78, -2.91]
  Call Extruder 0.10645
  MoveL (T14285) to (103.84, 113.06, 15.9) mm, rotated rx 180 ry 0 rz -180 deg; joints [1.945, 71.319, -37.588, 3.499, -33.78, -2.91]
  Call Extruder 0.34896
  MoveL (T14286) to (111.94, 121.16, 15.9) mm, rotated rx 180 ry 0 rz -180 deg; joints [1.945, 71.319, -37.588, 3.499, -33.78, -2.91]
  Call Extruder 0.03385
  MoveL (T14287) to (113.06, 121.16, 15.9) mm, rotated rx 180 ry 0 rz -180 deg; joints [3.284, 67.968, -31.283, 5.486, -36.811, -4.397]
  Call Extruder 0.26588
  MoveL (T14288) to (119.23, 114.98, 15.9) mm, rotated rx 180 ry 0 rz -180 deg; joints [3.284, 67.968, -31.283, 5.486, -36.811, -4.397]
  Call Extruder 0.01104
  MoveL (T14289) to (119.23, 114.62, 15.9) mm, rotated rx 180 ry 0 rz -180 deg; joints [3.284, 67.968, -31.283, 5.486, -36.811, -4.397]
  Call Extruder 0.38239
  MoveL (T14290) to (110.35, 105.75, 15.9) mm, rotated rx 180 ry 0 rz -180 deg; joints [3.287, 67.811, -30.987, 5.474, -36.949, -4.38]
  Call Extruder 0.0094
  MoveL (T14291) to (110.04, 105.75, 15.9) mm, rotated rx 180 ry 0 rz -180 deg; joints [3.287, 67.811, -30.987, 5.474, -36.949, -4.38]
  Call Extruder 0.26705
  MoveL (T14292) to (103.84, 111.94, 15.9) mm, rotated rx 180 ry 0 rz -180 deg; joints [3.287, 67.811, -30.987, 5.474, -36.949, -4.38]
  Call Extruder 0.07441
  MoveL (T14293) to (103.84, 109.5, 15.9) mm, rotated rx 180 ry 0 rz -180 deg; joints [1.884, 71.313, -37.576, 3.389, -33.783, -2.818]
  Set speed (45.0 mm/s)
  Call Extruder -1.6
  MoveL (T14294) to (103.84, 109.5, 15.9) mm, rotated rx 180 ry 0 rz -180 deg; joints [1.884, 71.313, -37.576, 3.389, -33.783, -2.818]
  Set speed (120.0 mm/s)
  MoveL (T14295) to (103.84, 109.5, 15.9) mm, rotated rx 180 ry 0 rz -180 deg; joints [1.884, 71.313, -37.576, 3.389, -33.783, -2.818]
  Call Extruder -0.38
  MoveL (T14296) to (103.84, 110.57, 15.9) mm, rotated rx 180 ry 0 rz -180 deg; joints [1.823, 71.307, -37.565, 3.279, -33.785, -2.726]
  Set speed (45.0 mm/s)
  Call Extruder -0.02
  MoveL (T14297) to (103.84, 110.57, 15.9) mm, rotated rx 180 ry 0 rz -180 deg; joints [1.823, 71.307, -37.565, 3.279, -33.785, -2.726]
  Set speed (150.0 mm/s)
  MoveL (T14298) to (103.84, 110.57, 17.9) mm, rotated rx 180 ry 0 rz -180 deg; joints [3.291, 67.654, -30.693, 5.463, -37.087, -4.363]
  MoveL (T14299) to (119.81, 113.03, 17.9) mm, rotated rx 180 ry 0 rz -180 deg; joints [3.291, 67.654, -30.693, 5.463, -37.087, -4.363]
  MoveL (T14300) to (119.81, 113.03, 15.9) mm, rotated rx 180 ry 0 rz -180 deg; joints [3.291, 67.654, -30.693, 5.463, -37.087, -4.363]
  Set speed (40.0 mm/s)
  Call Extruder 2.0
  MoveL (T14301) to (119.81, 113.03, 15.9) mm, rotated rx 180 ry 0 rz -180 deg; joints [3.291, 67.654, -30.693, 5.463, -37.087, -4.363]
  Set speed (26.8 mm/s)
  MoveL (T14302) to (119.81, 113.03, 15.9) mm, rotated rx 180 ry 0 rz -180 deg; joints [3.295, 67.499, -30.401, 5.452, -37.223, -4.346]
  Call Extruder 0.04114
  MoveL (T14303) to (121.16, 113.04, 15.9) mm, rotated rx 180 ry 0 rz -180 deg; joints [3.295, 67.499, -30.401, 5.452, -37.223, -4.346]
  Call Extruder 0.03327
  MoveL (T14304) to (121.16, 111.94, 15.9) mm, rotated rx 180 ry 0 rz -180 deg; joints [3.295, 67.499, -30.401, 5.452, -37.223, -4.346]
  Call Extruder 0.04019
  MoveL (T14305) to (120.22, 111.01, 15.9) mm, rotated rx 180 ry 0 rz -180 deg; joints [1.762, 71.301, -37.555, 3.169, -33.787, -2.635]
  Call Extruder 0.02842
  MoveL (T14306) to (121.16, 111.01, 15.9) mm, rotated rx 180 ry 0 rz -180 deg; joints [1.762, 71.301, -37.555, 3.169, -33.787, -2.635]
  Call Extruder 0.02223
  MoveL (T14307) to (121.16, 111.74, 15.9) mm, rotated rx 180 ry 0 rz -180 deg; joints [1.701, 71.296, -37.544, 3.059, -33.789, -2.543]
  Set speed (150.0 mm/s)
  MoveL (T14308) to (121.02, 110.79, 15.9) mm, rotated rx 180 ry 0 rz -180 deg; joints [1.701, 71.296, -37.544, 3.059, -33.789, -2.543]
  Set speed (26.8 mm/s)
  MoveL (T14309) to (121.02, 110.79, 15.9) mm, rotated rx 180 ry 0 rz -180 deg; joints [1.701, 71.296, -37.544, 3.059, -33.789, -2.543]
  Call Extruder 0.01707
  MoveL (T14310) to (120.64, 110.42, 15.9) mm, rotated rx 180 ry 0 rz -180 deg; joints [3.298, 67.345, -30.111, 5.44, -37.359, -4.329]
  Call Extruder 0.01988
  MoveL (T14311) to (120.03, 110.42, 15.9) mm, rotated rx 180 ry 0 rz -180 deg; joints [3.302, 67.191, -29.822, 5.43, -37.494, -4.313]
  Call Extruder 0.00867
  MoveL (T14312) to (120.22, 110.6, 15.9) mm, rotated rx 180 ry 0 rz -180 deg; joints [3.302, 67.191, -29.822, 5.43, -37.494, -4.313]
  Call Extruder 0.01988
  MoveL (T14313) to (119.61, 110.61, 15.9) mm, rotated rx 180 ry 0 rz -180 deg; joints [3.302, 67.191, -29.822, 5.43, -37.494, -4.313]
  Call Extruder 0.01298
  MoveL (T14314) to (119.32, 110.32, 15.9) mm, rotated rx 180 ry 0 rz -180 deg; joints [3.302, 67.191, -29.822, 5.43, -37.494, -4.313]
  Set speed (45.0 mm/s)
  Call Extruder -1.6
  MoveL (T14315) to (119.32, 110.32, 15.9) mm, rotated rx 180 ry 0 rz -180 deg; joints [1.64, 71.29, -37.534, 2.949, -33.791, -2.452]
  Set speed (120.0 mm/s)
  MoveL (T14316) to (119.32, 110.32, 15.9) mm, rotated rx 180 ry 0 rz -180 deg; joints [1.64, 71.29, -37.534, 2.949, -33.791, -2.452]
  Call Extruder -0.14251
  MoveL (T14317) to (119.61, 110.61, 15.9) mm, rotated rx 180 ry 0 rz -180 deg; joints [1.64, 71.29, -37.534, 2.949, -33.791, -2.452]
  Call Extruder -0.21832
  MoveL (T14318) to (120.22, 110.6, 15.9) mm, rotated rx 180 ry 0 rz -180 deg; joints [1.64, 71.29, -37.534, 2.949, -33.791, -2.452]
  Call Extruder -0.01916
  MoveL (T14319) to (120.18, 110.57, 15.9) mm, rotated rx 180 ry 0 rz -180 deg; joints [1.579, 71.285, -37.525, 2.84, -33.793, -2.36]
  Set speed (45.0 mm/s)
  Call Extruder -0.02
  MoveL (T14320) to (120.18, 110.57, 15.9) mm, rotated rx 180 ry 0 rz -180 deg; joints [1.579, 71.285, -37.525, 2.84, -33.793, -2.36]
  Set speed (150.0 mm/s)
  MoveL (T14321) to (120.18, 110.57, 17.9) mm, rotated rx 180 ry 0 rz -180 deg; joints [3.305, 67.039, -29.535, 5.419, -37.628, -4.297]
  MoveL (T14322) to (120.91, 113.79, 17.9) mm, rotated rx 180 ry 0 rz -180 deg; joints [3.305, 67.039, -29.535, 5.419, -37.628, -4.297]
  MoveL (T14323) to (120.91, 113.79, 15.9) mm, rotated rx 180 ry 0 rz -180 deg; joints [3.309, 66.887, -29.249, 5.409, -37.761, -4.281]
  Set speed (40.0 mm/s)
  Call Extruder 2.0
  MoveL (T14324) to (120.91, 113.79, 15.9) mm, rotated rx 180 ry 0 rz -180 deg; joints [3.309, 66.887, -29.249, 5.409, -37.761, -4.281]
  Set speed (26.8 mm/s)
  MoveL (T14325) to (120.91, 113.79, 15.9) mm, rotated rx 180 ry 0 rz -180 deg; joints [3.309, 66.887, -29.249, 5.409, -37.761, -4.281]
  Call Extruder 0.01625
  MoveL (T14326) to (120.56, 113.44, 15.9) mm, rotated rx 180 ry 0 rz -180 deg; joints [1.518, 71.28, -37.516, 2.73, -33.795, -2.269]
  Call Extruder 0.02044
  MoveL (T14327) to (119.94, 113.44, 15.9) mm, rotated rx 180 ry 0 rz -180 deg; joints [1.518, 71.28, -37.516, 2.73, -33.795, -2.269]
  Call Extruder 0.01625
  MoveL (T14328) to (120.29, 113.79, 15.9) mm, rotated rx 180 ry 0 rz -180 deg; joints [1.457, 71.276, -37.507, 2.62, -33.797, -2.178]
  Set speed (45.0 mm/s)
  Call Extruder -1.6
  MoveL (T14329) to (120.29, 113.79, 15.9) mm, rotated rx 180 ry 0 rz -180 deg; joints [1.457, 71.276, -37.507, 2.62, -33.797, -2.178]
  Set speed (120.0 mm/s)
  MoveL (T14330) to (120.29, 113.79, 15.9) mm, rotated rx 180 ry 0 rz -180 deg; joints [3.313, 66.736, -28.966, 5.398, -37.894, -4.265]
  Call Extruder -0.17616
  MoveL (T14331) to (119.94, 113.44, 15.9) mm, rotated rx 180 ry 0 rz -180 deg; joints [3.313, 66.736, -28.966, 5.398, -37.894, -4.265]
  Call Extruder -0.20384
  MoveL (T14332) to (120.51, 113.44, 15.9) mm, rotated rx 180 ry 0 rz -180 deg; joints [3.313, 66.736, -28.966, 5.398, -37.894, -4.265]
  Set speed (45.0 mm/s)
  Call Extruder -0.02
  MoveL (T14333) to (120.51, 113.44, 15.9) mm, rotated rx 180 ry 0 rz -180 deg; joints [3.316, 66.586, -28.683, 5.388, -38.026, -4.249]
  Set speed (150.0 mm/s)
  MoveL (T14334) to (120.51, 113.44, 17.9) mm, rotated rx 180 ry 0 rz -180 deg; joints [3.316, 66.586, -28.683, 5.388, -38.026, -4.249]
  MoveL (T14335) to (104.34, 103.54, 17.9) mm, rotated rx 180 ry 0 rz -180 deg; joints [1.396, 71.271, -37.498, 2.51, -33.799, -2.086]
  MoveL (T14336) to (104.34, 103.54, 16.1) mm, rotated rx 180 ry 0 rz -180 deg; joints [1.396, 71.271, -37.498, 2.51, -33.799, -2.086]
  Set speed (40.0 mm/s)
  Call Extruder 2.0
  MoveL (T14337) to (104.34, 103.54, 16.1) mm, rotated rx 180 ry 0 rz -180 deg; joints [1.397, 71.09, -37.158, 2.502, -33.958, -2.076]
  Call Extruder 0.52159
  MoveL (T14338) to (121.46, 103.54, 16.1) mm, rotated rx 180 ry 0 rz -180 deg; joints [1.397, 71.09, -37.158, 2.502, -33.958, -2.076]
  Call Extruder 0.31948
  MoveL (T14339) to (121.46, 114.03, 16.1) mm, rotated rx 180 ry 0 rz -180 deg; joints [1.397, 71.09, -37.158, 2.502, -33.958, -2.076]
  Call Extruder 0.05873
  MoveL (T14340) to (119.53, 114.02, 16.1) mm, rotated rx 180 ry 0 rz -180 deg; joints [3.253, 66.577, -28.667, 5.286, -38.029, -4.168]
  Call Extruder 0.11571
  MoveL (T14341) to (119.53, 117.82, 16.1) mm, rotated rx 180 ry 0 rz -180 deg; joints [3.253, 66.577, -28.667, 5.286, -38.029, -4.168]
  Call Extruder 0.05878
  MoveL (T14342) to (121.46, 117.83, 16.1) mm, rotated rx 180 ry 0 rz -180 deg; joints [3.253, 66.577, -28.667, 5.286, -38.029, -4.168]
  Call Extruder 0.11078
  MoveL (T14343) to (121.46, 121.46, 16.1) mm, rotated rx 180 ry 0 rz -180 deg; joints [3.253, 66.577, -28.667, 5.286, -38.029, -4.168]
  Call Extruder 0.54596
  MoveL (T14344) to (103.54, 121.46, 16.1) mm, rotated rx 180 ry 0 rz -180 deg; joints [3.253, 66.577, -28.667, 5.286, -38.029, -4.168]
  Call Extruder 0.54596
  MoveL (T14345) to (103.54, 103.54, 16.1) mm, rotated rx 180 ry 0 rz -180 deg; joints [3.191, 66.569, -28.651, 5.183, -38.031, -4.087]
  Call Extruder 0.02254
  MoveL (T14346) to (104.28, 103.54, 16.1) mm, rotated rx 180 ry 0 rz -180 deg; joints [3.191, 66.569, -28.651, 5.183, -38.031, -4.087]
  Set speed (150.0 mm/s)
  MoveL (T14347) to (103.53, 103.13, 16.1) mm, rotated rx 180 ry 0 rz -180 deg; joints [3.191, 66.569, -28.651, 5.183, -38.031, -4.087]
  Set speed (40.0 mm/s)
  MoveL (T14348) to (103.53, 103.13, 16.1) mm, rotated rx 180 ry 0 rz -180 deg; joints [1.399, 70.911, -36.821, 2.495, -34.115, -2.066]
  Call Extruder 0.55858
  MoveL (T14349) to (121.87, 103.13, 16.1) mm, rotated rx 180 ry 0 rz -180 deg; joints [1.399, 70.911, -36.821, 2.495, -34.115, -2.066]
  Call Extruder 0.3443
  MoveL (T14350) to (121.87, 114.43, 16.1) mm, rotated rx 180 ry 0 rz -180 deg; joints [1.399, 70.911, -36.821, 2.495, -34.115, -2.066]
  Call Extruder 0.05873
  MoveL (T14351) to (119.94, 114.43, 16.1) mm, rotated rx 180 ry 0 rz -180 deg; joints [1.4, 70.733, -36.486, 2.487, -34.272, -2.056]
  Call Extruder 0.0909
  MoveL (T14352) to (119.94, 117.42, 16.1) mm, rotated rx 180 ry 0 rz -180 deg; joints [1.4, 70.733, -36.486, 2.487, -34.272, -2.056]
  Call Extruder 0.05877
  MoveL (T14353) to (121.87, 117.42, 16.1) mm, rotated rx 180 ry 0 rz -180 deg; joints [1.4, 70.733, -36.486, 2.487, -34.272, -2.056]
  Call Extruder 0.13556
  MoveL (T14354) to (121.87, 121.87, 16.1) mm, rotated rx 180 ry 0 rz -180 deg; joints [3.128, 66.561, -28.636, 5.081, -38.034, -4.006]
  Call Extruder 0.57077
  MoveL (T14355) to (103.13, 121.87, 16.1) mm, rotated rx 180 ry 0 rz -180 deg; joints [3.128, 66.561, -28.636, 5.081, -38.034, -4.006]
  Call Extruder 0.57077
  MoveL (T14356) to (103.13, 103.13, 16.1) mm, rotated rx 180 ry 0 rz -180 deg; joints [3.128, 66.561, -28.636, 5.081, -38.034, -4.006]
  Call Extruder 0.01036
  MoveL (T14357) to (103.47, 103.13, 16.1) mm, rotated rx 180 ry 0 rz -180 deg; joints [3.065, 66.553, -28.621, 4.978, -38.037, -3.925]
  Set speed (150.0 mm/s)
  MoveL (T14358) to (102.72, 102.81, 16.1) mm, rotated rx 180 ry 0 rz -180 deg; joints [3.065, 66.553, -28.621, 4.978, -38.037, -3.925]
  Set speed (25.0 mm/s)
  MoveL (T14359) to (102.72, 102.81, 16.1) mm, rotated rx 180 ry 0 rz -180 deg; joints [1.402, 70.557, -36.154, 2.48, -34.428, -2.046]
  Call Extruder 0.00259
  MoveL (T14360) to (102.72, 102.72, 16.1) mm, rotated rx 180 ry 0 rz -180 deg; joints [1.402, 70.557, -36.154, 2.48, -34.428, -2.046]
  Call Extruder 0.59557
  MoveL (T14361) to (122.28, 102.72, 16.1) mm, rotated rx 180 ry 0 rz -180 deg; joints [1.402, 70.557, -36.154, 2.48, -34.428, -2.046]
  Call Extruder 0.36912
  MoveL (T14362) to (122.28, 114.84, 16.1) mm, rotated rx 180 ry 0 rz -180 deg; joints [1.403, 70.382, -35.825, 2.473, -34.582, -2.037]
  Call Extruder 0.05874
  MoveL (T14363) to (120.35, 114.84, 16.1) mm, rotated rx 180 ry 0 rz -180 deg; joints [1.403, 70.382, -35.825, 2.473, -34.582, -2.037]
  Call Extruder 0.0661
  MoveL (T14364) to (120.35, 117.01, 16.1) mm, rotated rx 180 ry 0 rz -180 deg; joints [1.403, 70.382, -35.825, 2.473, -34.582, -2.037]
  Call Extruder 0.05877
  MoveL (T14365) to (122.28, 117.01, 16.1) mm, rotated rx 180 ry 0 rz -180 deg; joints [3.002, 66.545, -28.606, 4.876, -38.04, -3.843]
  Call Extruder 0.16035
  MoveL (T14366) to (122.28, 122.28, 16.1) mm, rotated rx 180 ry 0 rz -180 deg; joints [3.002, 66.545, -28.606, 4.876, -38.04, -3.843]
  Call Extruder 0.59557
  MoveL (T14367) to (102.72, 122.28, 16.1) mm, rotated rx 180 ry 0 rz -180 deg; joints [3.002, 66.545, -28.606, 4.876, -38.04, -3.843]
  Call Extruder 0.59115
  MoveL (T14368) to (102.72, 102.87, 16.1) mm, rotated rx 180 ry 0 rz -180 deg; joints [3.002, 66.545, -28.606, 4.876, -38.04, -3.843]
  Set speed (150.0 mm/s)
  MoveL (T14369) to (102.78, 102.75, 16.1) mm, rotated rx 180 ry 0 rz -180 deg; joints [2.939, 66.537, -28.591, 4.773, -38.042, -3.762]
  Set speed (45.0 mm/s)
  Call Extruder -1.6
  MoveL (T14370) to (102.78, 102.75, 16.1) mm, rotated rx 180 ry 0 rz -180 deg; joints [2.939, 66.537, -28.591, 4.773, -38.042, -3.762]
  Set speed (120.0 mm/s)
  MoveL (T14371) to (102.78, 102.75, 16.1) mm, rotated rx 180 ry 0 rz -180 deg; joints [1.405, 70.208, -35.498, 2.466, -34.735, -2.027]
  Call Extruder -0.05166
  MoveL (T14372) to (102.72, 102.72, 16.1) mm, rotated rx 180 ry 0 rz -180 deg; joints [1.405, 70.208, -35.498, 2.466, -34.735, -2.027]
  Call Extruder -0.32834
  MoveL (T14373) to (103.65, 102.72, 16.1) mm, rotated rx 180 ry 0 rz -180 deg; joints [1.405, 70.208, -35.498, 2.466, -34.735, -2.027]
  Set speed (45.0 mm/s)
  Call Extruder -0.02
  MoveL (T14374) to (103.65, 102.72, 16.1) mm, rotated rx 180 ry 0 rz -180 deg; joints [1.406, 70.036, -35.174, 2.46, -34.887, -2.018]
  Set speed (150.0 mm/s)
  MoveL (T14375) to (103.65, 102.72, 18.1) mm, rotated rx 180 ry 0 rz -180 deg; joints [1.406, 70.036, -35.174, 2.46, -34.887, -2.018]
  MoveL (T14376) to (103.84, 106.29, 18.1) mm, rotated rx 180 ry 0 rz -180 deg; joints [2.876, 66.529, -28.577, 4.671, -38.045, -3.681]
  MoveL (T14377) to (103.84, 106.29, 16.1) mm, rotated rx 180 ry 0 rz -180 deg; joints [2.876, 66.529, -28.577, 4.671, -38.045, -3.681]
  Set speed (40.0 mm/s)
  Call Extruder 2.0
  MoveL (T14378) to (103.84, 106.29, 16.1) mm, rotated rx 180 ry 0 rz -180 deg; joints [2.813, 66.522, -28.563, 4.568, -38.047, -3.6]
  Set speed (50.0 mm/s)
  MoveL (T14379) to (103.84, 106.29, 16.1) mm, rotated rx 180 ry 0 rz -180 deg; joints [2.813, 66.522, -28.563, 4.568, -38.047, -3.6]
  Call Extruder 0.07441
  MoveL (T14380) to (103.84, 103.84, 16.1) mm, rotated rx 180 ry 0 rz -180 deg; joints [2.813, 66.522, -28.563, 4.568, -38.047, -3.6]
  Call Extruder 0.03503
  MoveL (T14381) to (104.66, 104.66, 16.1) mm, rotated rx 180 ry 0 rz -180 deg; joints [1.408, 69.865, -34.852, 2.453, -35.038, -2.009]
  Call Extruder 0.03259
  MoveL (T14382) to (104.66, 105.73, 16.1) mm, rotated rx 180 ry 0 rz -180 deg; joints [1.408, 69.865, -34.852, 2.453, -35.038, -2.009]
  Call Extruder 0.01721
  MoveL (T14383) to (105.06, 106.13, 16.1) mm, rotated rx 180 ry 0 rz -180 deg; joints [1.408, 69.865, -34.852, 2.453, -35.038, -2.009]
  Call Extruder 0.05221
  MoveL (T14384) to (103.84, 107.34, 16.1) mm, rotated rx 180 ry 0 rz -180 deg; joints [1.408, 69.865, -34.852, 2.453, -35.038, -2.009]
  Call Extruder 0.03385
  MoveL (T14385) to (103.84, 108.45, 16.1) mm, rotated rx 180 ry 0 rz -180 deg; joints [1.409, 69.695, -34.532, 2.446, -35.187, -2]
  Call Extruder 0.54738
  MoveL (T14386) to (116.55, 121.16, 16.1) mm, rotated rx 180 ry 0 rz -180 deg; joints [2.751, 66.515, -28.549, 4.466, -38.05, -3.519]
  Call Extruder 0.03385
  MoveL (T14387) to (117.66, 121.16, 16.1) mm, rotated rx 180 ry 0 rz -180 deg; joints [2.751, 66.515, -28.549, 4.466, -38.05, -3.519]
  Call Extruder 0.1304
  MoveL (T14388) to (120.69, 118.13, 16.1) mm, rotated rx 180 ry 0 rz -180 deg; joints [2.751, 66.515, -28.549, 4.466, -38.05, -3.519]
  Call Extruder 0.01425
  MoveL (T14389) to (121.16, 118.13, 16.1) mm, rotated rx 180 ry 0 rz -180 deg; joints [2.751, 66.515, -28.549, 4.466, -38.05, -3.519]
  Call Extruder 0.09219
  MoveL (T14390) to (121.16, 121.16, 16.1) mm, rotated rx 180 ry 0 rz -180 deg; joints [2.688, 66.508, -28.536, 4.363, -38.052, -3.438]
  Call Extruder 0.58379
  MoveL (T14391) to (107.61, 107.61, 16.1) mm, rotated rx 180 ry 0 rz -180 deg; joints [2.688, 66.508, -28.536, 4.363, -38.052, -3.438]
  Call Extruder 0.01763
  MoveL (T14392) to (108.18, 107.61, 16.1) mm, rotated rx 180 ry 0 rz -180 deg; joints [1.411, 69.526, -34.215, 2.44, -35.336, -1.991]
  Call Extruder 0.18695
  MoveL (T14393) to (103.84, 111.94, 16.1) mm, rotated rx 180 ry 0 rz -180 deg; joints [1.411, 69.526, -34.215, 2.44, -35.336, -1.991]
  Call Extruder 0.03385
  MoveL (T14394) to (103.84, 113.06, 16.1) mm, rotated rx 180 ry 0 rz -180 deg; joints [1.412, 69.359, -33.899, 2.434, -35.484, -1.982]
  Call Extruder 0.34896
  MoveL (T14395) to (111.94, 121.16, 16.1) mm, rotated rx 180 ry 0 rz -180 deg; joints [1.412, 69.359, -33.899, 2.434, -35.484, -1.982]
  Call Extruder 0.03385
  MoveL (T14396) to (113.06, 121.16, 16.1) mm, rotated rx 180 ry 0 rz -180 deg; joints [1.412, 69.359, -33.899, 2.434, -35.484, -1.982]
  Call Extruder 0.26589
  MoveL (T14397) to (119.23, 114.98, 16.1) mm, rotated rx 180 ry 0 rz -180 deg; joints [2.625, 66.501, -28.523, 4.261, -38.055, -3.357]
  Call Extruder 0.01102
  MoveL (T14398) to (119.23, 114.62, 16.1) mm, rotated rx 180 ry 0 rz -180 deg; joints [2.625, 66.501, -28.523, 4.261, -38.055, -3.357]
  Call Extruder 0.33185
  MoveL (T14399) to (111.53, 106.92, 16.1) mm, rotated rx 180 ry 0 rz -180 deg; joints [2.562, 66.494, -28.51, 4.158, -38.057, -3.276]
  Call Extruder 0.02835
  MoveL (T14400) to (112.18, 106.26, 16.1) mm, rotated rx 180 ry 0 rz -180 deg; joints [1.414, 69.192, -33.586, 2.428, -35.63, -1.974]
  Call Extruder 0.042
  MoveL (T14401) to (113.16, 107.24, 16.1) mm, rotated rx 180 ry 0 rz -180 deg; joints [1.414, 69.192, -33.586, 2.428, -35.63, -1.974]
  Call Extruder 0.40126
  MoveL (T14402) to (103.84, 116.55, 16.1) mm, rotated rx 180 ry 0 rz -180 deg; joints [1.416, 69.027, -33.276, 2.422, -35.775, -1.965]
  Call Extruder 0.03385
  MoveL (T14403) to (103.84, 117.66, 16.1) mm, rotated rx 180 ry 0 rz -180 deg; joints [1.416, 69.027, -33.276, 2.422, -35.775, -1.965]
  Call Extruder 0.15054
  MoveL (T14404) to (107.34, 121.16, 16.1) mm, rotated rx 180 ry 0 rz -180 deg; joints [2.499, 66.487, -28.498, 4.056, -38.059, -3.196]
  Call Extruder 0.03385
  MoveL (T14405) to (108.45, 121.16, 16.1) mm, rotated rx 180 ry 0 rz -180 deg; joints [2.499, 66.487, -28.498, 4.056, -38.059, -3.196]
  Call Extruder 0.42389
  MoveL (T14406) to (118.29, 111.32, 16.1) mm, rotated rx 180 ry 0 rz -180 deg; joints [2.499, 66.487, -28.498, 4.056, -38.059, -3.196]
  Call Extruder 0.0413
  MoveL (T14407) to (119.25, 112.28, 16.1) mm, rotated rx 180 ry 0 rz -180 deg; joints [2.436, 66.481, -28.486, 3.954, -38.061, -3.115]
  Call Extruder 0.05812
  MoveL (T14408) to (121.16, 112.27, 16.1) mm, rotated rx 180 ry 0 rz -180 deg; joints [2.436, 66.481, -28.486, 3.954, -38.061, -3.115]
  Call Extruder 0.02381
  MoveL (T14409) to (121.16, 113.06, 16.1) mm, rotated rx 180 ry 0 rz -180 deg; joints [1.417, 68.863, -32.967, 2.416, -35.92, -1.957]
  Call Extruder 0.00396
  MoveL (T14410) to (121.06, 113.15, 16.1) mm, rotated rx 180 ry 0 rz -180 deg; joints [1.417, 68.863, -32.967, 2.416, -35.92, -1.957]
  Call Extruder 0.05012
  MoveL (T14411) to (119.42, 113.14, 16.1) mm, rotated rx 180 ry 0 rz -180 deg; joints [1.417, 68.863, -32.967, 2.416, -35.92, -1.957]
  Call Extruder 0.01378
  MoveL (T14412) to (119.1, 113.47, 16.1) mm, rotated rx 180 ry 0 rz -180 deg; joints [1.419, 68.7, -32.661, 2.41, -36.064, -1.949]
  Call Extruder 0.01052
  MoveL (T14413) to (119.1, 113.81, 16.1) mm, rotated rx 180 ry 0 rz -180 deg; joints [1.419, 68.7, -32.661, 2.41, -36.064, -1.949]
  Set speed (150.0 mm/s)
  MoveL (T14414) to (121, 113.37, 16.1) mm, rotated rx 180 ry 0 rz -180 deg; joints [2.373, 66.475, -28.474, 3.851, -38.064, -3.034]
  Set speed (40.0 mm/s)
  MoveL (T14415) to (121, 113.37, 16.1) mm, rotated rx 180 ry 0 rz -180 deg; joints [2.373, 66.475, -28.474, 3.851, -38.064, -3.034]
  Call Extruder 0.01587
  MoveL (T14416) to (120.65, 113.72, 16.1) mm, rotated rx 180 ry 0 rz -180 deg; joints [2.373, 66.475, -28.474, 3.851, -38.064, -3.034]
  Call Extruder 0.01954
  MoveL (T14417) to (120.04, 113.72, 16.1) mm, rotated rx 180 ry 0 rz -180 deg; joints [2.31, 66.468, -28.462, 3.749, -38.066, -2.953]
  Call Extruder 0.00754
  MoveL (T14418) to (120.21, 113.55, 16.1) mm, rotated rx 180 ry 0 rz -180 deg; joints [2.31, 66.468, -28.462, 3.749, -38.066, -2.953]
  Call Extruder 0.01954
  MoveL (T14419) to (119.6, 113.55, 16.1) mm, rotated rx 180 ry 0 rz -180 deg; joints [2.31, 66.468, -28.462, 3.749, -38.066, -2.953]
  Call Extruder 0.01276
  MoveL (T14420) to (119.32, 113.83, 16.1) mm, rotated rx 180 ry 0 rz -180 deg; joints [1.42, 68.538, -32.356, 2.405, -36.206, -1.941]
  Set speed (45.0 mm/s)
  Call Extruder -1.6
  MoveL (T14421) to (119.32, 113.83, 16.1) mm, rotated rx 180 ry 0 rz -180 deg; joints [1.42, 68.538, -32.356, 2.405, -36.206, -1.941]
  Set speed (120.0 mm/s)
  MoveL (T14422) to (119.32, 113.83, 16.1) mm, rotated rx 180 ry 0 rz -180 deg; joints [1.42, 68.538, -32.356, 2.405, -36.206, -1.941]
  Call Extruder -0.14123
  MoveL (T14423) to (119.6, 113.55, 16.1) mm, rotated rx 180 ry 0 rz -180 deg; joints [1.422, 68.377, -32.053, 2.399, -36.348, -1.933]
  Call Extruder -0.21634
  MoveL (T14424) to (120.21, 113.55, 16.1) mm, rotated rx 180 ry 0 rz -180 deg; joints [1.422, 68.377, -32.053, 2.399, -36.348, -1.933]
  Call Extruder -0.02244
  MoveL (T14425) to (120.17, 113.6, 16.1) mm, rotated rx 180 ry 0 rz -180 deg; joints [2.247, 66.463, -28.451, 3.647, -38.068, -2.872]
  Set speed (45.0 mm/s)
  Call Extruder -0.02
  MoveL (T14426) to (120.17, 113.6, 16.1) mm, rotated rx 180 ry 0 rz -180 deg; joints [2.247, 66.463, -28.451, 3.647, -38.068, -2.872]
  Set speed (150.0 mm/s)
  MoveL (T14427) to (120.17, 113.6, 18.1) mm, rotated rx 180 ry 0 rz -180 deg; joints [2.247, 66.463, -28.451, 3.647, -38.068, -2.872]
  MoveL (T14428) to (114.37, 107.61, 18.1) mm, rotated rx 180 ry 0 rz -180 deg; joints [2.247, 66.463, -28.451, 3.647, -38.068, -2.872]
  MoveL (T14429) to (114.37, 107.61, 16.1) mm, rotated rx 180 ry 0 rz -180 deg; joints [2.185, 66.457, -28.44, 3.544, -38.07, -2.792]
  Set speed (40.0 mm/s)
  Call Extruder 2.0
  MoveL (T14430) to (114.37, 107.61, 16.1) mm, rotated rx 180 ry 0 rz -180 deg; joints [2.185, 66.457, -28.44, 3.544, -38.07, -2.792]
  Set speed (50.0 mm/s)
  MoveL (T14431) to (114.37, 107.61, 16.1) mm, rotated rx 180 ry 0 rz -180 deg; joints [2.185, 66.457, -28.44, 3.544, -38.07, -2.792]
  Call Extruder 0.07441
  MoveL (T14432) to (116.82, 107.61, 16.1) mm, rotated rx 180 ry 0 rz -180 deg; joints [1.423, 68.217, -31.752, 2.394, -36.489, -1.925]
  Call Extruder 0.0239
  MoveL (T14433) to (117.37, 108.16, 16.1) mm, rotated rx 180 ry 0 rz -180 deg; joints [1.423, 68.217, -31.752, 2.394, -36.489, -1.925]
  Call Extruder 0.01618
  MoveL (T14434) to (117.37, 107.63, 16.1) mm, rotated rx 180 ry 0 rz -180 deg; joints [1.425, 68.058, -31.453, 2.388, -36.629, -1.917]
  Call Extruder 0.58277
  MoveL (T14435) to (103.84, 121.16, 16.1) mm, rotated rx 180 ry 0 rz -180 deg; joints [1.425, 68.058, -31.453, 2.388, -36.629, -1.917]
  Call Extruder 0.07441
  MoveL (T14436) to (106.29, 121.16, 16.1) mm, rotated rx 180 ry 0 rz -180 deg; joints [1.425, 68.058, -31.453, 2.388, -36.629, -1.917]
  Set speed (45.0 mm/s)
  Call Extruder -1.6
  MoveL (T14437) to (106.29, 121.16, 16.1) mm, rotated rx 180 ry 0 rz -180 deg; joints [2.122, 66.451, -28.43, 3.442, -38.071, -2.711]
  Set speed (120.0 mm/s)
  MoveL (T14438) to (106.29, 121.16, 16.1) mm, rotated rx 180 ry 0 rz -180 deg; joints [2.122, 66.451, -28.43, 3.442, -38.071, -2.711]
  Call Extruder -0.38
  MoveL (T14439) to (105.22, 121.16, 16.1) mm, rotated rx 180 ry 0 rz -180 deg; joints [2.059, 66.446, -28.42, 3.34, -38.073, -2.63]
  Set speed (45.0 mm/s)
  Call Extruder -0.02
  MoveL (T14440) to (105.22, 121.16, 16.1) mm, rotated rx 180 ry 0 rz -180 deg; joints [2.059, 66.446, -28.42, 3.34, -38.073, -2.63]
  Set speed (150.0 mm/s)
  MoveL (T14441) to (105.22, 121.16, 18.1) mm, rotated rx 180 ry 0 rz -180 deg; joints [2.059, 66.446, -28.42, 3.34, -38.073, -2.63]
  MoveL (T14442) to (119.48, 103.82, 18.1) mm, rotated rx 180 ry 0 rz -180 deg; joints [1.426, 67.901, -31.156, 2.383, -36.768, -1.91]
  MoveL (T14443) to (119.48, 103.82, 16.1) mm, rotated rx 180 ry 0 rz -180 deg; joints [1.426, 67.901, -31.156, 2.383, -36.768, -1.91]
  Set speed (40.0 mm/s)
  Call Extruder 2.0
  MoveL (T14444) to (119.48, 103.82, 16.1) mm, rotated rx 180 ry 0 rz -180 deg; joints [1.428, 67.744, -30.861, 2.378, -36.906, -1.902]
  Set speed (25.0 mm/s)
  MoveL (T14445) to (119.48, 103.82, 16.1) mm, rotated rx 180 ry 0 rz -180 deg; joints [1.428, 67.744, -30.861, 2.378, -36.906, -1.902]
  Call Extruder 0.37984
  MoveL (T14446) to (105.03, 103.82, 16.1) mm, rotated rx 180 ry 0 rz -180 deg; joints [1.428, 67.744, -30.861, 2.378, -36.906, -1.902]
  Call Extruder 0.00923
  MoveL (T14447) to (105.03, 104.17, 16.1) mm, rotated rx 180 ry 0 rz -180 deg; joints [1.996, 66.44, -28.41, 3.237, -38.075, -2.549]
  Call Extruder 0.37576
  MoveL (T14448) to (119.33, 104.17, 16.1) mm, rotated rx 180 ry 0 rz -180 deg; joints [1.933, 66.435, -28.4, 3.135, -38.077, -2.469]
  Call Extruder 0.00886
  MoveL (T14449) to (119.33, 104.5, 16.1) mm, rotated rx 180 ry 0 rz -180 deg; joints [1.933, 66.435, -28.4, 3.135, -38.077, -2.469]
  Call Extruder 0.04882
  MoveL (T14450) to (121.19, 104.5, 16.1) mm, rotated rx 180 ry 0 rz -180 deg; joints [1.429, 67.588, -30.567, 2.373, -37.044, -1.895]
  Call Extruder 0.0004
  MoveL (T14451) to (121.19, 104.52, 16.1) mm, rotated rx 180 ry 0 rz -180 deg; joints [1.429, 67.588, -30.567, 2.373, -37.044, -1.895]
  Call Extruder 0.42459
  MoveL (T14452) to (105.03, 104.52, 16.1) mm, rotated rx 180 ry 0 rz -180 deg; joints [1.429, 67.588, -30.567, 2.373, -37.044, -1.895]
  Call Extruder 0.00923
  MoveL (T14453) to (105.03, 104.87, 16.1) mm, rotated rx 180 ry 0 rz -180 deg; joints [1.431, 67.432, -30.276, 2.368, -37.18, -1.887]
  Call Extruder 0.4246
  MoveL (T14454) to (121.19, 104.87, 16.1) mm, rotated rx 180 ry 0 rz -180 deg; joints [1.431, 67.432, -30.276, 2.368, -37.18, -1.887]
  Call Extruder 0.00923
  MoveL (T14455) to (121.19, 105.22, 16.1) mm, rotated rx 180 ry 0 rz -180 deg; joints [1.431, 67.432, -30.276, 2.368, -37.18, -1.887]
  Call Extruder 0.4246
  MoveL (T14456) to (105.03, 105.22, 16.1) mm, rotated rx 180 ry 0 rz -180 deg; joints [1.87, 66.43, -28.391, 3.033, -38.079, -2.388]
  Call Extruder 0.00923
  MoveL (T14457) to (105.03, 105.57, 16.1) mm, rotated rx 180 ry 0 rz -180 deg; joints [1.87, 66.43, -28.391, 3.033, -38.079, -2.388]
  Call Extruder 0.42457
  MoveL (T14458) to (121.19, 105.57, 16.1) mm, rotated rx 180 ry 0 rz -180 deg; joints [1.87, 66.43, -28.391, 3.033, -38.079, -2.388]
  Call Extruder 0.00923
  MoveL (T14459) to (121.19, 105.92, 16.1) mm, rotated rx 180 ry 0 rz -180 deg; joints [1.807, 66.426, -28.382, 2.93, -38.08, -2.307]
  Call Extruder 0.41534
  MoveL (T14460) to (105.39, 105.92, 16.1) mm, rotated rx 180 ry 0 rz -180 deg; joints [1.807, 66.426, -28.382, 2.93, -38.08, -2.307]
  Call Extruder 0.01306
  MoveL (T14461) to (105.74, 106.28, 16.1) mm, rotated rx 180 ry 0 rz -180 deg; joints [1.433, 67.278, -29.986, 2.364, -37.316, -1.88]
  Call Extruder 0.15507
  MoveL (T14462) to (111.64, 106.28, 16.1) mm, rotated rx 180 ry 0 rz -180 deg; joints [1.433, 67.278, -29.986, 2.364, -37.316, -1.88]
  Call Extruder 0.01306
  MoveL (T14463) to (111.28, 106.63, 16.1) mm, rotated rx 180 ry 0 rz -180 deg; joints [1.433, 67.278, -29.986, 2.364, -37.316, -1.88]
